LIN {X 0,Y 474.887,Z 291.332,A -85,B 0,C 180,E1 -7377.456,E2 -7377.456} C_VEL
LIN {X 0,Y 474.904,Z 291.328,A -85,B 0,C 180,E1 -7380,E2 -7380} C_VEL
LIN {X 0,Y 474.888,Z 291.326,A -85,B 0,C 180,E1 -7382.545,E2 -7382.545} C_VEL
LIN {X 0,Y 474.753,Z 291.35,A -85,B 0,C 180,E1 -7385.948,E2 -7385.948} C_VEL
LIN {X 0,Y 474.722,Z 291.348,A -85,B 0,C 180,E1 -7388.514,E2 -7388.514} C_VEL
LIN {X 0,Y 474.699,Z 291.357,A -85,B 0,C 180,E1 -7391.963,E2 -7391.963} C_VEL
LIN {X 0,Y 474.694,Z 291.35,A -85,B 0,C 180,E1 -7395.456,E2 -7395.456} C_VEL
LIN {X 0,Y 474.657,Z 291.355,A -85,B 0,C 180,E1 -7399.011,E2 -7399.011} C_VEL
LIN {X 0,Y 474.583,Z 291.365,A -85,B 0,C 180,E1 -7401.73,E2 -7401.73} C_VEL
LIN {X 0,Y 474.632,Z 291.365,A -85,B 0,C 180,E1 -7404.495,E2 -7404.495} C_VEL
LIN {X 0,Y 474.632,Z 291.357,A -85,B 0,C 180,E1 -7407.325,E2 -7407.325} C_VEL
LIN {X 0,Y 474.599,Z 291.366,A -85,B 0,C 180,E1 -7410.231,E2 -7410.231} C_VEL
LIN {X 0,Y 474.639,Z 291.358,A -85,B 0,C 180,E1 -7413.221,E2 -7413.221} C_VEL
LIN {X 0,Y 474.585,Z 291.367,A -85,B 0,C 180,E1 -7416.324,E2 -7416.324} C_VEL
LIN {X 0,Y 474.619,Z 291.359,A -85,B 0,C 180,E1 -7419.549,E2 -7419.549} C_VEL
LIN {X 0,Y 474.597,Z 291.363,A -85,B 0,C 180,E1 -7422.234,E2 -7422.234} C_VEL
LIN {X 0,Y 474.614,Z 291.364,A -85,B 0,C 180,E1 -7425.299,E2 -7425.299} C_VEL
LIN {X 0,Y 474.602,Z 291.361,A -85,B 0,C 180,E1 -7428.214,E2 -7428.214} C_VEL
LIN {X 0,Y 474.608,Z 291.363,A -85,B 0,C 180,E1 -7431.543,E2 -7431.543} C_VEL
LIN {X 0,Y 474.621,Z 291.361,A -85,B 0,C 180,E1 -7434.726,E2 -7434.726} C_VEL
LIN {X 0,Y 474.633,Z 291.359,A -85,B 0,C 180,E1 -7437.788,E2 -7437.788} C_VEL
LIN {X 0,Y 474.599,Z 291.364,A -85,B 0,C 180,E1 -7440.891,E2 -7440.891} C_VEL
LIN {X 0,Y 474.582,Z 291.37,A -85,B 0,C 180,E1 -7443.624,E2 -7443.624} C_VEL
LIN {X 0,Y 474.636,Z 291.357,A -85,B 0,C 180,E1 -7446.643,E2 -7446.643} C_VEL
LIN {X 0,Y 474.649,Z 291.358,A -85,B 0,C 180,E1 -7450.09,E2 -7450.09} C_VEL
LIN {X 0,Y 474.643,Z 291.361,A -85,B 0,C 180,E1 -7451.656,E2 -7451.656} C_VEL
LIN {X 0,Y 473.971,Z 291.446,A -85,B 0,C 180,E1 -7452.364,E2 -7452.364} C_VEL
LIN {X 0,Y 471.127,Z 291.8,A -85,B 0,C 180,E1 -7453.516,E2 -7453.516} C_VEL
LIN {X 0,Y 468.722,Z 292.097,A -85,B 0,C 180,E1 -7454.444,E2 -7454.444} C_VEL
LIN {X 0,Y 467.684,Z 292.224,A -85,B 0,C 180,E1 -7455.161,E2 -7455.161} C_VEL
LIN {X 0,Y 467.597,Z 292.235,A -85,B 0,C 180,E1 -7455.404,E2 -7455.404} C_VEL
LIN {X 0,Y 467.651,Z 292.236,A -85,B 0,C 180,E1 -7457.855,E2 -7457.855} C_VEL
LIN {X 0,Y 467.633,Z 292.231,A -85,B 0,C 180,E1 -7461.357,E2 -7461.357} C_VEL
LIN {X 0,Y 467.704,Z 292.229,A -85,B 0,C 180,E1 -7463.963,E2 -7463.963} C_VEL
LIN {X 0,Y 467.787,Z 292.211,A -85,B 0,C 180,E1 -7467.417,E2 -7467.417} C_VEL
LIN {X 0,Y 467.853,Z 292.208,A -85,B 0,C 180,E1 -7470.001,E2 -7470.001} C_VEL
LIN {X 0,Y 467.785,Z 292.214,A -85,B 0,C 180,E1 -7472.584,E2 -7472.584} C_VEL
LIN {X 0,Y 467.704,Z 292.225,A -85,B 0,C 180,E1 -7476.038,E2 -7476.038} C_VEL
LIN {X 0,Y 467.63,Z 292.235,A -85,B 0,C 180,E1 -7478.644,E2 -7478.644} C_VEL
LIN {X 0,Y 467.643,Z 292.234,A -85,B 0,C 180,E1 -7482.348,E2 -7482.348} C_VEL
LIN {X 0,Y 467.577,Z 292.237,A -85,B 0,C 180,E1 -7485.852,E2 -7485.852} C_VEL
LIN {X 0,Y 467.577,Z 292.245,A -85,B 0,C 180,E1 -7488.748,E2 -7488.748} C_VEL
LIN {X 0,Y 467.571,Z 292.242,A -85,B 0,C 180,E1 -7491.263,E2 -7491.263} C_VEL
LIN {X 0,Y 467.537,Z 292.245,A -85,B 0,C 180,E1 -7493.946,E2 -7493.946} C_VEL
LIN {X 0,Y 467.58,Z 292.359,A -85,B 0,C 180,E1 -7496.082,E2 -7496.082} C_VEL
LIN {X 0,Y 468.661,Z 298.553,A -85,B 0,C 180,E1 -7497.46,E2 -7497.46} C_VEL
LIN {X 0,Y 468.459,Z 309.115,A -85,B 0,C 180,E1 -7499.675,E2 -7499.675} C_VEL
LIN {X 0,Y 468.404,Z 311.167,A -85,B 0,C 180,E1 -7500.082,E2 -7500.082} C_VEL
LIN {X 0,Y 471.31,Z 326.35,A -85,B 0,C 180,E1 -7500.433,E2 -7500.433} C_VEL
LIN {X 0,Y 470.475,Z 418.507,A -85,B 0,C 180,E1 -7501.911,E2 -7501.911} C_VEL
LIN {X 0,Y 470.143,Z 431.815,A -85,B 0,C 180,E1 -7502.3,E2 -7502.3} C_VEL
LIN {X 0,Y 469.807,Z 444.646,A -85,B 0,C 180,E1 -7502.859,E2 -7502.859} C_VEL
LIN {X 0,Y 469.331,Z 456.478,A -85,B 0,C 180,E1 -7503.56,E2 -7503.56} C_VEL
LIN {X 0,Y 468.839,Z 468.329,A -85,B 0,C 180,E1 -7504.465,E2 -7504.465} C_VEL
LIN {X 0,Y 468.455,Z 478.228,A -85,B 0,C 180,E1 -7505.414,E2 -7505.414} C_VEL
LIN {X 0,Y 467.954,Z 487.6,A -85,B 0,C 180,E1 -7506.52,E2 -7506.52} C_VEL
LIN {X 0,Y 467.509,Z 496.556,A -85,B 0,C 180,E1 -7507.829,E2 -7507.829} C_VEL
LIN {X 0,Y 467.224,Z 503.935,A -85,B 0,C 180,E1 -7509.181,E2 -7509.181} C_VEL
LIN {X 0,Y 467.015,Z 508.97,A -85,B 0,C 180,E1 -7510.323,E2 -7510.323} C_VEL
LIN {X 0,Y 466.863,Z 513.083,A -85,B 0,C 180,E1 -7511.48,E2 -7511.48} C_VEL
LIN {X 0,Y 466.769,Z 516.363,A -85,B 0,C 180,E1 -7512.653,E2 -7512.653} C_VEL
LIN {X 0,Y 466.666,Z 518.873,A -85,B 0,C 180,E1 -7513.849,E2 -7513.849} C_VEL
LIN {X 0,Y 466.591,Z 520.607,A -85,B 0,C 180,E1 -7515.067,E2 -7515.067} C_VEL
LIN {X 0,Y 466.532,Z 521.536,A -85,B 0,C 180,E1 -7516.31,E2 -7516.31} C_VEL
LIN {X 0,Y 466.543,Z 521.611,A -85,B 0,C 180,E1 -7517.573,E2 -7517.573} C_VEL
LIN {X 0,Y 466.574,Z 520.813,A -85,B 0,C 180,E1 -7518.864,E2 -7518.864} C_VEL
LIN {X 0,Y 466.622,Z 519.065,A -85,B 0,C 180,E1 -7520.187,E2 -7520.187} C_VEL
LIN {X 0,Y 466.819,Z 515.392,A -85,B 0,C 180,E1 -7521.883,E2 -7521.883} C_VEL
LIN {X 0,Y 467.001,Z 510.099,A -85,B 0,C 180,E1 -7523.526,E2 -7523.526} C_VEL
LIN {X 0,Y 467.215,Z 504.977,A -85,B 0,C 180,E1 -7524.744,E2 -7524.744} C_VEL
LIN {X 0,Y 467.512,Z 498.452,A -85,B 0,C 180,E1 -7525.997,E2 -7525.997} C_VEL
LIN {X 0,Y 467.921,Z 490.267,A -85,B 0,C 180,E1 -7527.268,E2 -7527.268} C_VEL
LIN {X 0,Y 468.382,Z 480.754,A -85,B 0,C 180,E1 -7528.452,E2 -7528.452} C_VEL
LIN {X 0,Y 468.826,Z 470.415,A -85,B 0,C 180,E1 -7529.494,E2 -7529.494} C_VEL
LIN {X 0,Y 469.328,Z 459.314,A -85,B 0,C 180,E1 -7530.385,E2 -7530.385} C_VEL
LIN {X 0,Y 469.751,Z 447.055,A -85,B 0,C 180,E1 -7531.151,E2 -7531.151} C_VEL
LIN {X 0,Y 470.146,Z 434.659,A -85,B 0,C 180,E1 -7531.731,E2 -7531.731} C_VEL
LIN {X 0,Y 470.41,Z 422.487,A -85,B 0,C 180,E1 -7532.126,E2 -7532.126} C_VEL
LIN {X 0,Y 470.633,Z 405.056,A -85,B 0,C 180,E1 -7532.454,E2 -7532.454} C_VEL
LIN {X 0,Y 471.418,Z 326.13,A -85,B 0,C 180,E1 -7533.712,E2 -7533.712} C_VEL
LIN {X 0,Y 468.44,Z 310.387,A -85,B 0,C 180,E1 -7534.11,E2 -7534.11} C_VEL
LIN {X 0,Y 468.588,Z 297.583,A -85,B 0,C 180,E1 -7536.338,E2 -7536.338} C_VEL
LIN {X 0,Y 467.613,Z 292.241,A -85,B 0,C 180,E1 -7537.348,E2 -7537.348} C_VEL
LIN {X 0,Y 467.624,Z 292.236,A -85,B 0,C 180,E1 -7540.692,E2 -7540.692} C_VEL
LIN {X 0,Y 467.652,Z 292.233,A -85,B 0,C 180,E1 -7544.115,E2 -7544.115} C_VEL
LIN {X 0,Y 467.656,Z 292.235,A -85,B 0,C 180,E1 -7547.642,E2 -7547.642} C_VEL
LIN {X 0,Y 467.662,Z 292.228,A -85,B 0,C 180,E1 -7550.485,E2 -7550.485} C_VEL
LIN {X 0,Y 467.702,Z 292.224,A -85,B 0,C 180,E1 -7553.095,E2 -7553.095} C_VEL
LIN {X 0,Y 467.722,Z 292.221,A -85,B 0,C 180,E1 -7554.827,E2 -7554.827} C_VEL
LIN {X 0,Y 467.86,Z 292.206,A -85,B 0,C 180,E1 -7557.417,E2 -7557.417} C_VEL
LIN {X 0,Y 467.884,Z 292.205,A -85,B 0,C 180,E1 -7560,E2 -7560} C_VEL
LIN {X 0,Y 467.861,Z 292.204,A -85,B 0,C 180,E1 -7562.583,E2 -7562.583} C_VEL
LIN {X 0,Y 467.722,Z 292.226,A -85,B 0,C 180,E1 -7566.037,E2 -7566.037} C_VEL
LIN {X 0,Y 467.682,Z 292.227,A -85,B 0,C 180,E1 -7568.643,E2 -7568.643} C_VEL
LIN {X 0,Y 467.657,Z 292.233,A -85,B 0,C 180,E1 -7572.145,E2 -7572.145} C_VEL
LIN {X 0,Y 467.641,Z 292.23,A -85,B 0,C 180,E1 -7575.695,E2 -7575.695} C_VEL
LIN {X 0,Y 467.614,Z 292.238,A -85,B 0,C 180,E1 -7578.763,E2 -7578.763} C_VEL
LIN {X 0,Y 467.582,Z 292.236,A -85,B 0,C 180,E1 -7581.268,E2 -7581.268} C_VEL
LIN {X 0,Y 467.573,Z 292.237,A -85,B 0,C 180,E1 -7583.943,E2 -7583.943} C_VEL
LIN {X 0,Y 467.619,Z 292.238,A -85,B 0,C 180,E1 -7586.8,E2 -7586.8} C_VEL
LIN {X 0,Y 467.556,Z 292.24,A -85,B 0,C 180,E1 -7589.738,E2 -7589.738} C_VEL
LIN {X 0,Y 467.58,Z 292.24,A -85,B 0,C 180,E1 -7592.759,E2 -7592.759} C_VEL
LIN {X 0,Y 467.554,Z 292.241,A -85,B 0,C 180,E1 -7595.89,E2 -7595.89} C_VEL
LIN {X 0,Y 467.577,Z 292.244,A -85,B 0,C 180,E1 -7599.145,E2 -7599.145} C_VEL
LIN {X 0,Y 467.588,Z 292.238,A -85,B 0,C 180,E1 -7602.567,E2 -7602.567} C_VEL
LIN {X 0,Y 467.568,Z 292.244,A -85,B 0,C 180,E1 -7605.052,E2 -7605.052} C_VEL
LIN {X 0,Y 467.591,Z 292.243,A -85,B 0,C 180,E1 -7607.44,E2 -7607.44} C_VEL
LIN {X 0,Y 467.562,Z 292.241,A -85,B 0,C 180,E1 -7610.853,E2 -7610.853} C_VEL
LIN {X 0,Y 467.562,Z 292.245,A -85,B 0,C 180,E1 -7614.261,E2 -7614.261} C_VEL
LIN {X 0,Y 467.584,Z 292.244,A -85,B 0,C 180,E1 -7617.321,E2 -7617.321} C_VEL
LIN {X 0,Y 467.572,Z 292.241,A -85,B 0,C 180,E1 -7620.667,E2 -7620.667} C_VEL
LIN {X 0,Y 467.62,Z 292.239,A -85,B 0,C 180,E1 -7623.2,E2 -7623.2} C_VEL
LIN {X 0,Y 467.666,Z 292.395,A -85,B 0,C 180,E1 -7624.28,E2 -7624.28} C_VEL
LIN {X 0,Y 469.569,Z 302.744,A -85,B 0,C 180,E1 -7626.164,E2 -7626.164} C_VEL
LIN {X 0,Y 469.161,Z 316.935,A -85,B 0,C 180,E1 -7628.572,E2 -7628.572} C_VEL
LIN {X 0,Y 468.509,Z 336.543,A -85,B 0,C 180,E1 -7631.864,E2 -7631.864} C_VEL
LIN {X 0,Y 468.238,Z 342.994,A -85,B 0,C 180,E1 -7632.938,E2 -7632.938} C_VEL
LIN {X 0,Y 471.17,Z 362.703,A -85,B 0,C 180,E1 -7633.383,E2 -7633.383} C_VEL
LIN {X 0,Y 470.398,Z 451.756,A -85,B 0,C 180,E1 -7634.815,E2 -7634.815} C_VEL
LIN {X 0,Y 470.029,Z 464.941,A -85,B 0,C 180,E1 -7635.191,E2 -7635.191} C_VEL
LIN {X 0,Y 469.56,Z 478.23,A -85,B 0,C 180,E1 -7635.757,E2 -7635.757} C_VEL
LIN {X 0,Y 469.065,Z 490.218,A -85,B 0,C 180,E1 -7636.46,E2 -7636.46} C_VEL
LIN {X 0,Y 468.579,Z 502.383,A -85,B 0,C 180,E1 -7637.384,E2 -7637.384} C_VEL
LIN {X 0,Y 468.155,Z 512.119,A -85,B 0,C 180,E1 -7638.307,E2 -7638.307} C_VEL
LIN {X 0,Y 467.67,Z 521.451,A -85,B 0,C 180,E1 -7639.392,E2 -7639.392} C_VEL
LIN {X 0,Y 467.255,Z 530.522,A -85,B 0,C 180,E1 -7640.694,E2 -7640.694} C_VEL
LIN {X 0,Y 467.009,Z 537.837,A -85,B 0,C 180,E1 -7641.998,E2 -7641.998} C_VEL
LIN {X 0,Y 466.842,Z 542.78,A -85,B 0,C 180,E1 -7643.082,E2 -7643.082} C_VEL
LIN {X 0,Y 466.76,Z 547.587,A -85,B 0,C 180,E1 -7644.383,E2 -7644.383} C_VEL
LIN {X 0,Y 466.647,Z 551.26,A -85,B 0,C 180,E1 -7645.681,E2 -7645.681} C_VEL
LIN {X 0,Y 466.69,Z 553.16,A -85,B 0,C 180,E1 -7646.546,E2 -7646.546} C_VEL
LIN {X 0,Y 466.662,Z 554.584,A -85,B 0,C 180,E1 -7647.41,E2 -7647.41} C_VEL
LIN {X 0,Y 466.619,Z 556.227,A -85,B 0,C 180,E1 -7649.137,E2 -7649.137} C_VEL
LIN {X 0,Y 466.6,Z 556.451,A -85,B 0,C 180,E1 -7649.999,E2 -7649.999} C_VEL
LIN {X 0,Y 466.619,Z 556.237,A -85,B 0,C 180,E1 -7650.862,E2 -7650.862} C_VEL
LIN {X 0,Y 466.661,Z 554.626,A -85,B 0,C 180,E1 -7652.589,E2 -7652.589} C_VEL
LIN {X 0,Y 466.689,Z 553.211,A -85,B 0,C 180,E1 -7653.453,E2 -7653.453} C_VEL
LIN {X 0,Y 466.689,Z 550.24,A -85,B 0,C 180,E1 -7654.75,E2 -7654.75} C_VEL
LIN {X 0,Y 466.749,Z 546.214,A -85,B 0,C 180,E1 -7656.05,E2 -7656.05} C_VEL
LIN {X 0,Y 466.94,Z 540.011,A -85,B 0,C 180,E1 -7657.567,E2 -7657.567} C_VEL
LIN {X 0,Y 467.163,Z 533.24,A -85,B 0,C 180,E1 -7658.87,E2 -7658.87} C_VEL
LIN {X 0,Y 467.498,Z 524.835,A -85,B 0,C 180,E1 -7660.174,E2 -7660.174} C_VEL
LIN {X 0,Y 467.938,Z 516.177,A -85,B 0,C 180,E1 -7661.259,E2 -7661.259} C_VEL
LIN {X 0,Y 468.442,Z 505.997,A -85,B 0,C 180,E1 -7662.299,E2 -7662.299} C_VEL
LIN {X 0,Y 468.887,Z 494.923,A -85,B 0,C 180,E1 -7663.213,E2 -7663.213} C_VEL
LIN {X 0,Y 469.35,Z 483.182,A -85,B 0,C 180,E1 -7663.972,E2 -7663.972} C_VEL
LIN {X 0,Y 469.832,Z 470.995,A -85,B 0,C 180,E1 -7664.565,E2 -7664.565} C_VEL
LIN {X 0,Y 470.213,Z 457.736,A -85,B 0,C 180,E1 -7665.024,E2 -7665.024} C_VEL
LIN {X 0,Y 470.478,Z 443.027,A -85,B 0,C 180,E1 -7665.32,E2 -7665.32} C_VEL
LIN {X 0,Y 471.075,Z 362.031,A -85,B 0,C 180,E1 -7666.602,E2 -7666.602} C_VEL
LIN {X 0,Y 468.31,Z 343.777,A -85,B 0,C 180,E1 -7667.016,E2 -7667.016} C_VEL
LIN {X 0,Y 468.981,Z 326.897,A -85,B 0,C 180,E1 -7669.933,E2 -7669.933} C_VEL
LIN {X 0,Y 469.808,Z 309.995,A -85,B 0,C 180,E1 -7672.888,E2 -7672.888} C_VEL
LIN {X 0,Y 469.753,Z 303.092,A -85,B 0,C 180,E1 -7674.129,E2 -7674.129} C_VEL
LIN {X 0,Y 467.649,Z 292.236,A -85,B 0,C 180,E1 -7676.226,E2 -7676.226} C_VEL
LIN {X 0,Y 467.569,Z 292.24,A -85,B 0,C 180,E1 -7679.332,E2 -7679.332} C_VEL
LIN {X 0,Y 467.58,Z 292.239,A -85,B 0,C 180,E1 -7682.678,E2 -7682.678} C_VEL
LIN {X 0,Y 467.557,Z 292.241,A -85,B 0,C 180,E1 -7685.738,E2 -7685.738} C_VEL
LIN {X 0,Y 467.557,Z 292.239,A -85,B 0,C 180,E1 -7689.146,E2 -7689.146} C_VEL
LIN {X 0,Y 467.583,Z 292.242,A -85,B 0,C 180,E1 -7692.566,E2 -7692.566} C_VEL
LIN {X 0,Y 467.567,Z 292.239,A -85,B 0,C 180,E1 -7695.053,E2 -7695.053} C_VEL
LIN {X 0,Y 467.585,Z 292.235,A -85,B 0,C 180,E1 -7697.439,E2 -7697.439} C_VEL
LIN {X 0,Y 467.578,Z 292.242,A -85,B 0,C 180,E1 -7700.855,E2 -7700.855} C_VEL
LIN {X 0,Y 467.558,Z 292.241,A -85,B 0,C 180,E1 -7704.26,E2 -7704.26} C_VEL
LIN {X 0,Y 467.577,Z 292.239,A -85,B 0,C 180,E1 -7707.32,E2 -7707.32} C_VEL
LIN {X 0,Y 467.565,Z 292.243,A -85,B 0,C 180,E1 -7710.667,E2 -7710.667} C_VEL
LIN {X 0,Y 467.611,Z 292.238,A -85,B 0,C 180,E1 -7713.199,E2 -7713.199} C_VEL
LIN {X 0,Y 467.587,Z 292.236,A -85,B 0,C 180,E1 -7716.468,E2 -7716.468} C_VEL
LIN {X 0,Y 467.617,Z 292.233,A -85,B 0,C 180,E1 -7719.777,E2 -7719.777} C_VEL
LIN {X 0,Y 467.603,Z 292.234,A -85,B 0,C 180,E1 -7722.507,E2 -7722.507} C_VEL
LIN {X 0,Y 467.604,Z 292.24,A -85,B 0,C 180,E1 -7725.196,E2 -7725.196} C_VEL
LIN {X 0,Y 467.65,Z 292.23,A -85,B 0,C 180,E1 -7727.855,E2 -7727.855} C_VEL
LIN {X 0,Y 467.676,Z 292.231,A -85,B 0,C 180,E1 -7731.357,E2 -7731.357} C_VEL
LIN {X 0,Y 467.737,Z 292.219,A -85,B 0,C 180,E1 -7733.963,E2 -7733.963} C_VEL
LIN {X 0,Y 467.853,Z 292.207,A -85,B 0,C 180,E1 -7737.417,E2 -7737.417} C_VEL
LIN {X 0,Y 467.875,Z 292.204,A -85,B 0,C 180,E1 -7740,E2 -7740} C_VEL
LIN {X 0,Y 467.853,Z 292.202,A -85,B 0,C 180,E1 -7742.583,E2 -7742.583} C_VEL
LIN {X 0,Y 467.716,Z 292.226,A -85,B 0,C 180,E1 -7746.038,E2 -7746.038} C_VEL
LIN {X 0,Y 467.676,Z 292.225,A -85,B 0,C 180,E1 -7748.643,E2 -7748.643} C_VEL
LIN {X 0,Y 467.65,Z 292.235,A -85,B 0,C 180,E1 -7752.146,E2 -7752.146} C_VEL
LIN {X 0,Y 467.633,Z 292.232,A -85,B 0,C 180,E1 -7755.696,E2 -7755.696} C_VEL
LIN {X 0,Y 467.617,Z 292.231,A -85,B 0,C 180,E1 -7759.308,E2 -7759.308} C_VEL
LIN {X 0,Y 467.529,Z 292.247,A -85,B 0,C 180,E1 -7762.074,E2 -7762.074} C_VEL
LIN {X 0,Y 467.578,Z 292.238,A -85,B 0,C 180,E1 -7764.889,E2 -7764.889} C_VEL
LIN {X 0,Y 467.575,Z 292.237,A -85,B 0,C 180,E1 -7767.772,E2 -7767.772} C_VEL
LIN {X 0,Y 467.564,Z 292.24,A -85,B 0,C 180,E1 -7771.046,E2 -7771.046} C_VEL
LIN {X 0,Y 467.585,Z 292.238,A -85,B 0,C 180,E1 -7774.243,E2 -7774.243} C_VEL
LIN {X 0,Y 467.544,Z 292.243,A -85,B 0,C 180,E1 -7777.187,E2 -7777.187} C_VEL
LIN {X 0,Y 467.566,Z 292.239,A -85,B 0,C 180,E1 -7780.266,E2 -7780.266} C_VEL
LIN {X 0,Y 467.558,Z 292.243,A -85,B 0,C 180,E1 -7782.564,E2 -7782.564} C_VEL
LIN {X 0,Y 467.564,Z 292.245,A -85,B 0,C 180,E1 -7785.053,E2 -7785.053} C_VEL
LIN {X 0,Y 467.564,Z 292.242,A -85,B 0,C 180,E1 -7788.726,E2 -7788.726} C_VEL
LIN {X 0,Y 467.562,Z 292.238,A -85,B 0,C 180,E1 -7791.956,E2 -7791.956} C_VEL
LIN {X 0,Y 467.558,Z 292.247,A -85,B 0,C 180,E1 -7795.168,E2 -7795.168} C_VEL
LIN {X 0,Y 467.58,Z 292.236,A -85,B 0,C 180,E1 -7798.261,E2 -7798.261} C_VEL
LIN {X 0,Y 467.546,Z 292.247,A -85,B 0,C 180,E1 -7801.249,E2 -7801.249} C_VEL
LIN {X 0,Y 467.577,Z 292.236,A -85,B 0,C 180,E1 -7804.402,E2 -7804.402} C_VEL
LIN {X 0,Y 467.578,Z 292.238,A -85,B 0,C 180,E1 -7806.997,E2 -7806.997} C_VEL
LIN {X 0,Y 467.62,Z 292.237,A -85,B 0,C 180,E1 -7809.778,E2 -7809.778} C_VEL
LIN {X 0,Y 467.589,Z 292.235,A -85,B 0,C 180,E1 -7812.507,E2 -7812.507} C_VEL
LIN {X 0,Y 467.597,Z 292.235,A -85,B 0,C 180,E1 -7815.404,E2 -7815.404} C_VEL
LIN {X 0,Y 466.924,Z 292.322,A -85,B 0,C 180,E1 -7816.123,E2 -7816.123} C_VEL
LIN {X 0,Y 464.076,Z 292.674,A -85,B 0,C 180,E1 -7817.291,E2 -7817.291} C_VEL
LIN {X 0,Y 461.671,Z 292.975,A -85,B 0,C 180,E1 -7818.233,E2 -7818.233} C_VEL
LIN {X 0,Y 460.638,Z 293.101,A -85,B 0,C 180,E1 -7818.961,E2 -7818.961} C_VEL
LIN {X 0,Y 460.553,Z 293.112,A -85,B 0,C 180,E1 -7819.207,E2 -7819.207} C_VEL
LIN {X 0,Y 460.667,Z 293.098,A -85,B 0,C 180,E1 -7822.595,E2 -7822.595} C_VEL
LIN {X 0,Y 460.676,Z 293.097,A -85,B 0,C 180,E1 -7824.749,E2 -7824.749} C_VEL
LIN {X 0,Y 460.718,Z 293.098,A -85,B 0,C 180,E1 -7828.252,E2 -7828.252} C_VEL
LIN {X 0,Y 460.822,Z 293.084,A -85,B 0,C 180,E1 -7830.001,E2 -7830.001} C_VEL
LIN {X 0,Y 460.732,Z 293.092,A -85,B 0,C 180,E1 -7832.623,E2 -7832.623} C_VEL
LIN {X 0,Y 460.67,Z 293.102,A -85,B 0,C 180,E1 -7836.131,E2 -7836.131} C_VEL
LIN {X 0,Y 460.584,Z 293.111,A -85,B 0,C 180,E1 -7838.777,E2 -7838.777} C_VEL
LIN {X 0,Y 460.602,Z 293.113,A -85,B 0,C 180,E1 -7842.435,E2 -7842.435} C_VEL
LIN {X 0,Y 460.531,Z 293.115,A -85,B 0,C 180,E1 -7845.965,E2 -7845.965} C_VEL
LIN {X 0,Y 460.535,Z 293.121,A -85,B 0,C 180,E1 -7848.887,E2 -7848.887} C_VEL
LIN {X 0,Y 460.516,Z 293.119,A -85,B 0,C 180,E1 -7851.486,E2 -7851.486} C_VEL
LIN {X 0,Y 460.5,Z 293.124,A -85,B 0,C 180,E1 -7854.335,E2 -7854.335} C_VEL
LIN {X 0,Y 460.551,Z 293.198,A -85,B 0,C 180,E1 -7855.904,E2 -7855.904} C_VEL
LIN {X 0,Y 461.786,Z 300.731,A -85,B 0,C 180,E1 -7857.593,E2 -7857.593} C_VEL
LIN {X 0,Y 461.463,Z 311.503,A -85,B 0,C 180,E1 -7859.83,E2 -7859.83} C_VEL
LIN {X 0,Y 464.48,Z 327.191,A -85,B 0,C 180,E1 -7860.203,E2 -7860.203} C_VEL
LIN {X 0,Y 463.601,Z 418.569,A -85,B 0,C 180,E1 -7861.692,E2 -7861.692} C_VEL
LIN {X 0,Y 463.247,Z 431.996,A -85,B 0,C 180,E1 -7862.089,E2 -7862.089} C_VEL
LIN {X 0,Y 462.943,Z 443.935,A -85,B 0,C 180,E1 -7862.611,E2 -7862.611} C_VEL
LIN {X 0,Y 462.456,Z 455.653,A -85,B 0,C 180,E1 -7863.296,E2 -7863.296} C_VEL
LIN {X 0,Y 461.964,Z 466.743,A -85,B 0,C 180,E1 -7864.132,E2 -7864.132} C_VEL
LIN {X 0,Y 461.501,Z 477.687,A -85,B 0,C 180,E1 -7865.168,E2 -7865.168} C_VEL
LIN {X 0,Y 461.043,Z 486.998,A -85,B 0,C 180,E1 -7866.26,E2 -7866.26} C_VEL
LIN {X 0,Y 460.569,Z 495.479,A -85,B 0,C 180,E1 -7867.487,E2 -7867.487} C_VEL
LIN {X 0,Y 460.21,Z 503.066,A -85,B 0,C 180,E1 -7868.845,E2 -7868.845} C_VEL
LIN {X 0,Y 459.948,Z 509.024,A -85,B 0,C 180,E1 -7870.181,E2 -7870.181} C_VEL
LIN {X 0,Y 459.786,Z 513.638,A -85,B 0,C 180,E1 -7871.497,E2 -7871.497} C_VEL
LIN {X 0,Y 459.67,Z 517.091,A -85,B 0,C 180,E1 -7872.786,E2 -7872.786} C_VEL
LIN {X 0,Y 459.552,Z 519.529,A -85,B 0,C 180,E1 -7874.046,E2 -7874.046} C_VEL
LIN {X 0,Y 459.484,Z 521.091,A -85,B 0,C 180,E1 -7875.284,E2 -7875.284} C_VEL
LIN {X 0,Y 459.438,Z 521.856,A -85,B 0,C 180,E1 -7876.499,E2 -7876.499} C_VEL
LIN {X 0,Y 459.447,Z 521.859,A -85,B 0,C 180,E1 -7877.696,E2 -7877.696} C_VEL
LIN {X 0,Y 459.485,Z 521.102,A -85,B 0,C 180,E1 -7878.875,E2 -7878.875} C_VEL
LIN {X 0,Y 459.53,Z 519.676,A -85,B 0,C 180,E1 -7880.033,E2 -7880.033} C_VEL
LIN {X 0,Y 459.649,Z 517.422,A -85,B 0,C 180,E1 -7881.241,E2 -7881.241} C_VEL
LIN {X 0,Y 459.819,Z 513.752,A -85,B 0,C 180,E1 -7882.635,E2 -7882.635} C_VEL
LIN {X 0,Y 460.028,Z 508.693,A -85,B 0,C 180,E1 -7884.067,E2 -7884.067} C_VEL
LIN {X 0,Y 460.36,Z 501.626,A -85,B 0,C 180,E1 -7885.607,E2 -7885.607} C_VEL
LIN {X 0,Y 460.813,Z 493.323,A -85,B 0,C 180,E1 -7887.016,E2 -7887.016} C_VEL
LIN {X 0,Y 461.253,Z 484.363,A -85,B 0,C 180,E1 -7888.235,E2 -7888.235} C_VEL
LIN {X 0,Y 461.72,Z 474.342,A -85,B 0,C 180,E1 -7889.341,E2 -7889.341} C_VEL
LIN {X 0,Y 462.234,Z 463.584,A -85,B 0,C 180,E1 -7890.287,E2 -7890.287} C_VEL
LIN {X 0,Y 462.769,Z 451.178,A -85,B 0,C 180,E1 -7891.146,E2 -7891.146} C_VEL
LIN {X 0,Y 463.192,Z 439.482,A -85,B 0,C 180,E1 -7891.76,E2 -7891.76} C_VEL
LIN {X 0,Y 463.466,Z 425.92,A -85,B 0,C 180,E1 -7892.267,E2 -7892.267} C_VEL
LIN {X 0,Y 463.76,Z 412.27,A -85,B 0,C 180,E1 -7892.577,E2 -7892.577} C_VEL
LIN {X 0,Y 464.586,Z 326.297,A -85,B 0,C 180,E1 -7893.979,E2 -7893.979} C_VEL
LIN {X 0,Y 461.528,Z 310.691,A -85,B 0,C 180,E1 -7894.378,E2 -7894.378} C_VEL
LIN {X 0,Y 461.687,Z 299.498,A -85,B 0,C 180,E1 -7896.34,E2 -7896.34} C_VEL
LIN {X 0,Y 460.556,Z 293.119,A -85,B 0,C 180,E1 -7897.544,E2 -7897.544} C_VEL
LIN {X 0,Y 460.571,Z 293.113,A -85,B 0,C 180,E1 -7900.384,E2 -7900.384} C_VEL
LIN {X 0,Y 460.603,Z 293.112,A -85,B 0,C 180,E1 -7904.002,E2 -7904.002} C_VEL
LIN {X 0,Y 460.611,Z 293.112,A -85,B 0,C 180,E1 -7907.666,E2 -7907.666} C_VEL
LIN {X 0,Y 460.628,Z 293.107,A -85,B 0,C 180,E1 -7911.224,E2 -7911.224} C_VEL
LIN {X 0,Y 460.702,Z 293.1,A -85,B 0,C 180,E1 -7913.87,E2 -7913.87} C_VEL
LIN {X 0,Y 460.801,Z 293.085,A -85,B 0,C 180,E1 -7917.377,E2 -7917.377} C_VEL
LIN {X 0,Y 460.854,Z 293.081,A -85,B 0,C 180,E1 -7920,E2 -7920} C_VEL
LIN {X 0,Y 460.802,Z 293.083,A -85,B 0,C 180,E1 -7922.622,E2 -7922.622} C_VEL
LIN {X 0,Y 460.686,Z 293.101,A -85,B 0,C 180,E1 -7926.13,E2 -7926.13} C_VEL
LIN {X 0,Y 460.629,Z 293.104,A -85,B 0,C 180,E1 -7928.776,E2 -7928.776} C_VEL
LIN {X 0,Y 460.615,Z 293.109,A -85,B 0,C 180,E1 -7932.445,E2 -7932.445} C_VEL
LIN {X 0,Y 460.602,Z 293.109,A -85,B 0,C 180,E1 -7935.997,E2 -7935.997} C_VEL
LIN {X 0,Y 460.569,Z 293.11,A -85,B 0,C 180,E1 -7939.615,E2 -7939.615} C_VEL
LIN {X 0,Y 460.512,Z 293.121,A -85,B 0,C 180,E1 -7942.429,E2 -7942.429} C_VEL
LIN {X 0,Y 460.569,Z 293.109,A -85,B 0,C 180,E1 -7945.802,E2 -7945.802} C_VEL
LIN {X 0,Y 460.554,Z 293.109,A -85,B 0,C 180,E1 -7948.233,E2 -7948.233} C_VEL
LIN {X 0,Y 460.522,Z 293.118,A -85,B 0,C 180,E1 -7951.283,E2 -7951.283} C_VEL
LIN {X 0,Y 460.524,Z 293.117,A -85,B 0,C 180,E1 -7954.504,E2 -7954.504} C_VEL
LIN {X 0,Y 460.503,Z 293.119,A -85,B 0,C 180,E1 -7957.623,E2 -7957.623} C_VEL
LIN {X 0,Y 460.541,Z 293.113,A -85,B 0,C 180,E1 -7960.269,E2 -7960.269} C_VEL
LIN {X 0,Y 460.501,Z 293.124,A -85,B 0,C 180,E1 -7963.375,E2 -7963.375} C_VEL
LIN {X 0,Y 460.5,Z 293.12,A -85,B 0,C 180,E1 -7966.624,E2 -7966.624} C_VEL
LIN {X 0,Y 460.541,Z 293.119,A -85,B 0,C 180,E1 -7969.731,E2 -7969.731} C_VEL
LIN {X 0,Y 460.502,Z 293.122,A -85,B 0,C 180,E1 -7972.524,E2 -7972.524} C_VEL
LIN {X 0,Y 460.549,Z 293.123,A -85,B 0,C 180,E1 -7975.624,E2 -7975.624} C_VEL
LIN {X 0,Y 460.54,Z 293.117,A -85,B 0,C 180,E1 -7978.744,E2 -7978.744} C_VEL
LIN {X 0,Y 460.584,Z 293.116,A -85,B 0,C 180,E1 -7982.254,E2 -7982.254} C_VEL
LIN {X 0,Y 460.614,Z 293.192,A -85,B 0,C 180,E1 -7984.045,E2 -7984.045} C_VEL
LIN {X 0,Y 462.538,Z 303.263,A -85,B 0,C 180,E1 -7985.922,E2 -7985.922} C_VEL
LIN {X 0,Y 462.622,Z 307.903,A -85,B 0,C 180,E1 -7986.735,E2 -7986.735} C_VEL
LIN {X 0,Y 461.894,Z 326.853,A -85,B 0,C 180,E1 -7989.979,E2 -7989.979} C_VEL
LIN {X 0,Y 461.277,Z 342.723,A -85,B 0,C 180,E1 -7992.666,E2 -7992.666} C_VEL
LIN {X 0,Y 464.368,Z 363.157,A -85,B 0,C 180,E1 -7993.133,E2 -7993.133} C_VEL
LIN {X 0,Y 463.564,Z 451.556,A -85,B 0,C 180,E1 -7994.586,E2 -7994.586} C_VEL
LIN {X 0,Y 463.176,Z 464.703,A -85,B 0,C 180,E1 -7994.967,E2 -7994.967} C_VEL
LIN {X 0,Y 462.658,Z 477.976,A -85,B 0,C 180,E1 -7995.54,E2 -7995.54} C_VEL
LIN {X 0,Y 462.145,Z 489.957,A -85,B 0,C 180,E1 -7996.254,E2 -7996.254} C_VEL
LIN {X 0,Y 461.66,Z 501.506,A -85,B 0,C 180,E1 -7997.139,E2 -7997.139} C_VEL
LIN {X 0,Y 461.183,Z 511.858,A -85,B 0,C 180,E1 -7998.127,E2 -7998.127} C_VEL
LIN {X 0,Y 460.639,Z 521.188,A -85,B 0,C 180,E1 -7999.228,E2 -7999.228} C_VEL
LIN {X 0,Y 460.209,Z 530.262,A -85,B 0,C 180,E1 -8000.551,E2 -8000.551} C_VEL
LIN {X 0,Y 459.95,Z 537.579,A -85,B 0,C 180,E1 -8001.874,E2 -8001.874} C_VEL
LIN {X 0,Y 459.74,Z 543.711,A -85,B 0,C 180,E1 -8003.272,E2 -8003.272} C_VEL
LIN {X 0,Y 459.65,Z 548.66,A -85,B 0,C 180,E1 -8004.736,E2 -8004.736} C_VEL
LIN {X 0,Y 459.565,Z 550.995,A -85,B 0,C 180,E1 -8005.614,E2 -8005.614} C_VEL
LIN {X 0,Y 459.585,Z 552.895,A -85,B 0,C 180,E1 -8006.493,E2 -8006.493} C_VEL
LIN {X 0,Y 459.584,Z 554.32,A -85,B 0,C 180,E1 -8007.37,E2 -8007.37} C_VEL
LIN {X 0,Y 459.552,Z 555.964,A -85,B 0,C 180,E1 -8009.123,E2 -8009.123} C_VEL
LIN {X 0,Y 459.532,Z 556.188,A -85,B 0,C 180,E1 -8009.999,E2 -8009.999} C_VEL
LIN {X 0,Y 459.552,Z 555.973,A -85,B 0,C 180,E1 -8010.876,E2 -8010.876} C_VEL
LIN {X 0,Y 459.584,Z 554.358,A -85,B 0,C 180,E1 -8012.629,E2 -8012.629} C_VEL
LIN {X 0,Y 459.585,Z 552.939,A -85,B 0,C 180,E1 -8013.506,E2 -8013.506} C_VEL
LIN {X 0,Y 459.616,Z 549.964,A -85,B 0,C 180,E1 -8014.824,E2 -8014.824} C_VEL
LIN {X 0,Y 459.713,Z 544.874,A -85,B 0,C 180,E1 -8016.43,E2 -8016.43} C_VEL
LIN {X 0,Y 459.889,Z 538.69,A -85,B 0,C 180,E1 -8017.905,E2 -8017.905} C_VEL
LIN {X 0,Y 460.175,Z 531.667,A -85,B 0,C 180,E1 -8019.227,E2 -8019.227} C_VEL
LIN {X 0,Y 460.557,Z 522.856,A -85,B 0,C 180,E1 -8020.551,E2 -8020.551} C_VEL
LIN {X 0,Y 461.119,Z 512.851,A -85,B 0,C 180,E1 -8021.762,E2 -8021.762} C_VEL
LIN {X 0,Y 461.561,Z 502.918,A -85,B 0,C 180,E1 -8022.732,E2 -8022.732} C_VEL
LIN {X 0,Y 462.069,Z 491.349,A -85,B 0,C 180,E1 -8023.635,E2 -8023.635} C_VEL
LIN {X 0,Y 462.561,Z 479.647,A -85,B 0,C 180,E1 -8024.349,E2 -8024.349} C_VEL
LIN {X 0,Y 463.046,Z 466.974,A -85,B 0,C 180,E1 -8024.924,E2 -8024.924} C_VEL
LIN {X 0,Y 463.466,Z 453.581,A -85,B 0,C 180,E1 -8025.332,E2 -8025.332} C_VEL
LIN {X 0,Y 463.809,Z 421.729,A -85,B 0,C 180,E1 -8025.871,E2 -8025.871} C_VEL
LIN {X 0,Y 464.197,Z 362.391,A -85,B 0,C 180,E1 -8026.833,E2 -8026.833} C_VEL
LIN {X 0,Y 461.324,Z 343.668,A -85,B 0,C 180,E1 -8027.249,E2 -8027.249} C_VEL
LIN {X 0,Y 462.074,Z 326.606,A -85,B 0,C 180,E1 -8030.243,E2 -8030.243} C_VEL
LIN {X 0,Y 462.965,Z 308.418,A -85,B 0,C 180,E1 -8033.483,E2 -8033.483} C_VEL
LIN {X 0,Y 462.61,Z 303.188,A -85,B 0,C 180,E1 -8034.454,E2 -8034.454} C_VEL
LIN {X 0,Y 460.587,Z 293.114,A -85,B 0,C 180,E1 -8036.446,E2 -8036.446} C_VEL
LIN {X 0,Y 460.53,Z 293.119,A -85,B 0,C 180,E1 -8039.558,E2 -8039.558} C_VEL
LIN {X 0,Y 460.53,Z 293.124,A -85,B 0,C 180,E1 -8042.284,E2 -8042.284} C_VEL
LIN {X 0,Y 460.508,Z 293.117,A -85,B 0,C 180,E1 -8045.445,E2 -8045.445} C_VEL
LIN {X 0,Y 460.531,Z 293.116,A -85,B 0,C 180,E1 -8048.895,E2 -8048.895} C_VEL
LIN {X 0,Y 460.519,Z 293.121,A -85,B 0,C 180,E1 -8052.181,E2 -8052.181} C_VEL
LIN {X 0,Y 460.517,Z 293.116,A -85,B 0,C 180,E1 -8055.411,E2 -8055.411} C_VEL
LIN {X 0,Y 460.531,Z 293.12,A -85,B 0,C 180,E1 -8058.396,E2 -8058.396} C_VEL
LIN {X 0,Y 460.523,Z 293.116,A -85,B 0,C 180,E1 -8061.267,E2 -8061.267} C_VEL
LIN {X 0,Y 460.508,Z 293.123,A -85,B 0,C 180,E1 -8064.554,E2 -8064.554} C_VEL
LIN {X 0,Y 460.527,Z 293.115,A -85,B 0,C 180,E1 -8067.715,E2 -8067.715} C_VEL
LIN {X 0,Y 460.535,Z 293.12,A -85,B 0,C 180,E1 -8070.769,E2 -8070.769} C_VEL
LIN {X 0,Y 460.558,Z 293.111,A -85,B 0,C 180,E1 -8073.734,E2 -8073.734} C_VEL
LIN {X 0,Y 460.54,Z 293.115,A -85,B 0,C 180,E1 -8076.624,E2 -8076.624} C_VEL
LIN {X 0,Y 460.545,Z 293.117,A -85,B 0,C 180,E1 -8079.453,E2 -8079.453} C_VEL
LIN {X 0,Y 460.553,Z 293.111,A -85,B 0,C 180,E1 -8082.23,E2 -8082.23} C_VEL
LIN {X 0,Y 460.562,Z 293.114,A -85,B 0,C 180,E1 -8084.965,E2 -8084.965} C_VEL
LIN {X 0,Y 460.605,Z 293.105,A -85,B 0,C 180,E1 -8088.559,E2 -8088.559} C_VEL
LIN {X 0,Y 460.689,Z 293.096,A -85,B 0,C 180,E1 -8092.109,E2 -8092.109} C_VEL
LIN {X 0,Y 460.69,Z 293.094,A -85,B 0,C 180,E1 -8094.748,E2 -8094.748} C_VEL
LIN {X 0,Y 460.793,Z 293.086,A -85,B 0,C 180,E1 -8097.378,E2 -8097.378} C_VEL
LIN {X 0,Y 460.845,Z 293.08,A -85,B 0,C 180,E1 -8100,E2 -8100} C_VEL
LIN {X 0,Y 460.794,Z 293.081,A -85,B 0,C 180,E1 -8102.623,E2 -8102.623} C_VEL
LIN {X 0,Y 460.68,Z 293.101,A -85,B 0,C 180,E1 -8106.131,E2 -8106.131} C_VEL
LIN {X 0,Y 460.623,Z 293.103,A -85,B 0,C 180,E1 -8108.777,E2 -8108.777} C_VEL
LIN {X 0,Y 460.608,Z 293.108,A -85,B 0,C 180,E1 -8112.445,E2 -8112.445} C_VEL
LIN {X 0,Y 460.595,Z 293.112,A -85,B 0,C 180,E1 -8115.998,E2 -8115.998} C_VEL
LIN {X 0,Y 460.563,Z 293.111,A -85,B 0,C 180,E1 -8119.616,E2 -8119.616} C_VEL
LIN {X 0,Y 460.506,Z 293.125,A -85,B 0,C 180,E1 -8122.429,E2 -8122.429} C_VEL
LIN {X 0,Y 460.544,Z 293.114,A -85,B 0,C 180,E1 -8125.798,E2 -8125.798} C_VEL
LIN {X 0,Y 460.522,Z 293.12,A -85,B 0,C 180,E1 -8128.235,E2 -8128.235} C_VEL
LIN {X 0,Y 460.517,Z 293.116,A -85,B 0,C 180,E1 -8131.284,E2 -8131.284} C_VEL
LIN {X 0,Y 460.528,Z 293.121,A -85,B 0,C 180,E1 -8134.506,E2 -8134.506} C_VEL
LIN {X 0,Y 460.497,Z 293.118,A -85,B 0,C 180,E1 -8137.624,E2 -8137.624} C_VEL
LIN {X 0,Y 460.531,Z 293.116,A -85,B 0,C 180,E1 -8140.269,E2 -8140.269} C_VEL
LIN {X 0,Y 460.506,Z 293.12,A -85,B 0,C 180,E1 -8143.375,E2 -8143.375} C_VEL
LIN {X 0,Y 460.501,Z 293.121,A -85,B 0,C 180,E1 -8146.626,E2 -8146.626} C_VEL
LIN {X 0,Y 460.523,Z 293.116,A -85,B 0,C 180,E1 -8149.734,E2 -8149.734} C_VEL
LIN {X 0,Y 460.498,Z 293.119,A -85,B 0,C 180,E1 -8152.525,E2 -8152.525} C_VEL
LIN {X 0,Y 460.537,Z 293.117,A -85,B 0,C 180,E1 -8155.624,E2 -8155.624} C_VEL
LIN {X 0,Y 460.521,Z 293.117,A -85,B 0,C 180,E1 -8158.744,E2 -8158.744} C_VEL
LIN {X 0,Y 460.508,Z 293.12,A -85,B 0,C 180,E1 -8161.765,E2 -8161.765} C_VEL
LIN {X 0,Y 460.521,Z 293.116,A -85,B 0,C 180,E1 -8164.704,E2 -8164.704} C_VEL
LIN {X 0,Y 460.513,Z 293.125,A -85,B 0,C 180,E1 -8167.572,E2 -8167.572} C_VEL
LIN {X 0,Y 460.567,Z 293.11,A -85,B 0,C 180,E1 -8170.385,E2 -8170.385} C_VEL
LIN {X 0,Y 460.582,Z 293.112,A -85,B 0,C 180,E1 -8174.013,E2 -8174.013} C_VEL
LIN {X 0,Y 460.606,Z 293.111,A -85,B 0,C 180,E1 -8177.666,E2 -8177.666} C_VEL
LIN {X 0,Y 460.553,Z 293.112,A -85,B 0,C 180,E1 -8179.207,E2 -8179.207} C_VEL
LIN {X 0,Y 459.887,Z 293.203,A -85,B 0,C 180,E1 -8179.937,E2 -8179.937} C_VEL
LIN {X 0,Y 457.056,Z 293.55,A -85,B 0,C 180,E1 -8181.123,E2 -8181.123} C_VEL
LIN {X 0,Y 454.674,Z 293.851,A -85,B 0,C 180,E1 -8182.08,E2 -8182.08} C_VEL
LIN {X 0,Y 453.664,Z 293.97,A -85,B 0,C 180,E1 -8182.819,E2 -8182.819} C_VEL
LIN {X 0,Y 453.589,Z 293.979,A -85,B 0,C 180,E1 -8183.069,E2 -8183.069} C_VEL
LIN {X 0,Y 453.649,Z 293.972,A -85,B 0,C 180,E1 -8184.667,E2 -8184.667} C_VEL
LIN {X 0,Y 453.688,Z 293.974,A -85,B 0,C 180,E1 -8188.225,E2 -8188.225} C_VEL
LIN {X 0,Y 453.771,Z 293.962,A -85,B 0,C 180,E1 -8190.001,E2 -8190.001} C_VEL
LIN {X 0,Y 453.681,Z 293.97,A -85,B 0,C 180,E1 -8192.664,E2 -8192.664} C_VEL
LIN {X 0,Y 453.638,Z 293.98,A -85,B 0,C 180,E1 -8196.226,E2 -8196.226} C_VEL
LIN {X 0,Y 453.554,Z 293.985,A -85,B 0,C 180,E1 -8198.915,E2 -8198.915} C_VEL
LIN {X 0,Y 453.57,Z 293.99,A -85,B 0,C 180,E1 -8202.529,E2 -8202.529} C_VEL
LIN {X 0,Y 453.495,Z 293.993,A -85,B 0,C 180,E1 -8206.198,E2 -8206.198} C_VEL
LIN {X 0,Y 453.49,Z 293.997,A -85,B 0,C 180,E1 -8209.028,E2 -8209.028} C_VEL
LIN {X 0,Y 453.475,Z 293.996,A -85,B 0,C 180,E1 -8211.837,E2 -8211.837} C_VEL
LIN {X 0,Y 453.475,Z 294.001,A -85,B 0,C 180,E1 -8215.227,E2 -8215.227} C_VEL
LIN {X 0,Y 453.493,Z 294.029,A -85,B 0,C 180,E1 -8215.718,E2 -8215.718} C_VEL
LIN {X 0,Y 454.762,Z 301.294,A -85,B 0,C 180,E1 -8217.372,E2 -8217.372} C_VEL
LIN {X 0,Y 454.5,Z 311.538,A -85,B 0,C 180,E1 -8219.563,E2 -8219.563} C_VEL
LIN {X 0,Y 457.678,Z 328.34,A -85,B 0,C 180,E1 -8219.973,E2 -8219.973} C_VEL
LIN {X 0,Y 456.74,Z 419.157,A -85,B 0,C 180,E1 -8221.481,E2 -8221.481} C_VEL
LIN {X 0,Y 456.359,Z 432.62,A -85,B 0,C 180,E1 -8221.888,E2 -8221.888} C_VEL
LIN {X 0,Y 456.048,Z 444.203,A -85,B 0,C 180,E1 -8222.406,E2 -8222.406} C_VEL
LIN {X 0,Y 455.517,Z 456.548,A -85,B 0,C 180,E1 -8223.145,E2 -8223.145} C_VEL
LIN {X 0,Y 454.955,Z 468.228,A -85,B 0,C 180,E1 -8224.055,E2 -8224.055} C_VEL
LIN {X 0,Y 454.544,Z 477.636,A -85,B 0,C 180,E1 -8224.968,E2 -8224.968} C_VEL
LIN {X 0,Y 454.048,Z 486.658,A -85,B 0,C 180,E1 -8226.029,E2 -8226.029} C_VEL
LIN {X 0,Y 453.619,Z 494.647,A -85,B 0,C 180,E1 -8227.174,E2 -8227.174} C_VEL
LIN {X 0,Y 453.235,Z 502.32,A -85,B 0,C 180,E1 -8228.532,E2 -8228.532} C_VEL
LIN {X 0,Y 452.895,Z 508.934,A -85,B 0,C 180,E1 -8230.002,E2 -8230.002} C_VEL
LIN {X 0,Y 452.732,Z 513.344,A -85,B 0,C 180,E1 -8231.251,E2 -8231.251} C_VEL
LIN {X 0,Y 452.625,Z 516.763,A -85,B 0,C 180,E1 -8232.488,E2 -8232.488} C_VEL
LIN {X 0,Y 452.486,Z 519.318,A -85,B 0,C 180,E1 -8233.723,E2 -8233.723} C_VEL
LIN {X 0,Y 452.439,Z 520.36,A -85,B 0,C 180,E1 -8234.393,E2 -8234.393} C_VEL
LIN {X 0,Y 452.387,Z 521.693,A -85,B 0,C 180,E1 -8235.645,E2 -8235.645} C_VEL
LIN {X 0,Y 452.342,Z 522.201,A -85,B 0,C 180,E1 -8236.906,E2 -8236.906} C_VEL
LIN {X 0,Y 452.37,Z 521.882,A -85,B 0,C 180,E1 -8238.222,E2 -8238.222} C_VEL
LIN {X 0,Y 452.395,Z 520.652,A -85,B 0,C 180,E1 -8239.572,E2 -8239.572} C_VEL
LIN {X 0,Y 452.529,Z 518.435,A -85,B 0,C 180,E1 -8240.944,E2 -8240.944} C_VEL
LIN {X 0,Y 452.719,Z 515.101,A -85,B 0,C 180,E1 -8242.347,E2 -8242.347} C_VEL
LIN {X 0,Y 452.925,Z 510.179,A -85,B 0,C 180,E1 -8243.868,E2 -8243.868} C_VEL
LIN {X 0,Y 453.216,Z 504.246,A -85,B 0,C 180,E1 -8245.273,E2 -8245.273} C_VEL
LIN {X 0,Y 453.523,Z 497.968,A -85,B 0,C 180,E1 -8246.468,E2 -8246.468} C_VEL
LIN {X 0,Y 453.983,Z 489.904,A -85,B 0,C 180,E1 -8247.718,E2 -8247.718} C_VEL
LIN {X 0,Y 454.508,Z 480.263,A -85,B 0,C 180,E1 -8248.93,E2 -8248.93} C_VEL
LIN {X 0,Y 454.984,Z 470.963,A -85,B 0,C 180,E1 -8249.885,E2 -8249.885} C_VEL
LIN {X 0,Y 455.554,Z 459.929,A -85,B 0,C 180,E1 -8250.798,E2 -8250.798} C_VEL
LIN {X 0,Y 456.024,Z 448.262,A -85,B 0,C 180,E1 -8251.554,E2 -8251.554} C_VEL
LIN {X 0,Y 456.465,Z 435.467,A -85,B 0,C 180,E1 -8252.179,E2 -8252.179} C_VEL
LIN {X 0,Y 456.781,Z 422.76,A -85,B 0,C 180,E1 -8252.604,E2 -8252.604} C_VEL
LIN {X 0,Y 457.021,Z 405.311,A -85,B 0,C 180,E1 -8252.942,E2 -8252.942} C_VEL
LIN {X 0,Y 457.819,Z 327.03,A -85,B 0,C 180,E1 -8254.242,E2 -8254.242} C_VEL
LIN {X 0,Y 454.617,Z 310.814,A -85,B 0,C 180,E1 -8254.688,E2 -8254.688} C_VEL
LIN {X 0,Y 454.729,Z 300.361,A -85,B 0,C 180,E1 -8256.548,E2 -8256.548} C_VEL
LIN {X 0,Y 453.514,Z 293.995,A -85,B 0,C 180,E1 -8257.746,E2 -8257.746} C_VEL
LIN {X 0,Y 453.525,Z 293.996,A -85,B 0,C 180,E1 -8261.008,E2 -8261.008} C_VEL
LIN {X 0,Y 453.571,Z 293.989,A -85,B 0,C 180,E1 -8263.88,E2 -8263.88} C_VEL
LIN {X 0,Y 453.566,Z 293.991,A -85,B 0,C 180,E1 -8267.471,E2 -8267.471} C_VEL
LIN {X 0,Y 453.592,Z 293.983,A -85,B 0,C 180,E1 -8271.086,E2 -8271.086} C_VEL
LIN {X 0,Y 453.67,Z 293.976,A -85,B 0,C 180,E1 -8273.774,E2 -8273.774} C_VEL
LIN {X 0,Y 453.745,Z 293.964,A -85,B 0,C 180,E1 -8277.336,E2 -8277.336} C_VEL
LIN {X 0,Y 453.824,Z 293.956,A -85,B 0,C 180,E1 -8280,E2 -8280} C_VEL
LIN {X 0,Y 453.746,Z 293.961,A -85,B 0,C 180,E1 -8282.663,E2 -8282.663} C_VEL
LIN {X 0,Y 453.652,Z 293.975,A -85,B 0,C 180,E1 -8286.225,E2 -8286.225} C_VEL
LIN {X 0,Y 453.592,Z 293.98,A -85,B 0,C 180,E1 -8288.913,E2 -8288.913} C_VEL
LIN {X 0,Y 453.565,Z 293.986,A -85,B 0,C 180,E1 -8292.529,E2 -8292.529} C_VEL
LIN {X 0,Y 453.546,Z 293.991,A -85,B 0,C 180,E1 -8296.196,E2 -8296.196} C_VEL
LIN {X 0,Y 453.518,Z 293.991,A -85,B 0,C 180,E1 -8299.039,E2 -8299.039} C_VEL
LIN {X 0,Y 453.478,Z 293.992,A -85,B 0,C 180,E1 -8301.836,E2 -8301.836} C_VEL
LIN {X 0,Y 453.515,Z 293.991,A -85,B 0,C 180,E1 -8304.734,E2 -8304.734} C_VEL
LIN {X 0,Y 453.534,Z 293.983,A -85,B 0,C 180,E1 -8307.959,E2 -8307.959} C_VEL
LIN {X 0,Y 453.467,Z 293.995,A -85,B 0,C 180,E1 -8311.525,E2 -8311.525} C_VEL
LIN {X 0,Y 453.484,Z 293.996,A -85,B 0,C 180,E1 -8314.776,E2 -8314.776} C_VEL
LIN {X 0,Y 453.465,Z 293.994,A -85,B 0,C 180,E1 -8318.312,E2 -8318.312} C_VEL
LIN {X 0,Y 453.495,Z 293.992,A -85,B 0,C 180,E1 -8320.609,E2 -8320.609} C_VEL
LIN {X 0,Y 453.457,Z 294.002,A -85,B 0,C 180,E1 -8323.244,E2 -8323.244} C_VEL
LIN {X 0,Y 453.465,Z 293.999,A -85,B 0,C 180,E1 -8325.779,E2 -8325.779} C_VEL
LIN {X 0,Y 453.481,Z 293.994,A -85,B 0,C 180,E1 -8328.209,E2 -8328.209} C_VEL
LIN {X 0,Y 453.489,Z 293.994,A -85,B 0,C 180,E1 -8330.794,E2 -8330.794} C_VEL
LIN {X 0,Y 453.457,Z 294.006,A -85,B 0,C 180,E1 -8333.917,E2 -8333.917} C_VEL
LIN {X 0,Y 453.485,Z 294,A -85,B 0,C 180,E1 -8337.151,E2 -8337.151} C_VEL
LIN {X 0,Y 453.477,Z 293.999,A -85,B 0,C 180,E1 -8340.268,E2 -8340.268} C_VEL
LIN {X 0,Y 453.518,Z 293.997,A -85,B 0,C 180,E1 -8343.294,E2 -8343.294} C_VEL
LIN {X 0,Y 453.579,Z 294.174,A -85,B 0,C 180,E1 -8343.836,E2 -8343.836} C_VEL
LIN {X 0,Y 455.685,Z 305.35,A -85,B 0,C 180,E1 -8345.949,E2 -8345.949} C_VEL
LIN {X 0,Y 455.356,Z 316.797,A -85,B 0,C 180,E1 -8347.955,E2 -8347.955} C_VEL
LIN {X 0,Y 454.671,Z 334.714,A -85,B 0,C 180,E1 -8351.058,E2 -8351.058} C_VEL
LIN {X 0,Y 454.362,Z 342.373,A -85,B 0,C 180,E1 -8352.372,E2 -8352.372} C_VEL
LIN {X 0,Y 457.612,Z 364.665,A -85,B 0,C 180,E1 -8352.895,E2 -8352.895} C_VEL
LIN {X 0,Y 456.737,Z 451.482,A -85,B 0,C 180,E1 -8354.35,E2 -8354.35} C_VEL
LIN {X 0,Y 456.333,Z 464.528,A -85,B 0,C 180,E1 -8354.736,E2 -8354.736} C_VEL
LIN {X 0,Y 455.786,Z 477.746,A -85,B 0,C 180,E1 -8355.317,E2 -8355.317} C_VEL
LIN {X 0,Y 455.213,Z 489.696,A -85,B 0,C 180,E1 -8356.04,E2 -8356.04} C_VEL
LIN {X 0,Y 454.704,Z 501.244,A -85,B 0,C 180,E1 -8356.939,E2 -8356.939} C_VEL
LIN {X 0,Y 454.207,Z 511.597,A -85,B 0,C 180,E1 -8357.942,E2 -8357.942} C_VEL
LIN {X 0,Y 453.634,Z 520.926,A -85,B 0,C 180,E1 -8359.059,E2 -8359.059} C_VEL
LIN {X 0,Y 453.177,Z 530.004,A -85,B 0,C 180,E1 -8360.403,E2 -8360.403} C_VEL
LIN {X 0,Y 452.902,Z 537.323,A -85,B 0,C 180,E1 -8361.747,E2 -8361.747} C_VEL
LIN {X 0,Y 452.688,Z 542.261,A -85,B 0,C 180,E1 -8362.865,E2 -8362.865} C_VEL
LIN {X 0,Y 452.556,Z 547.066,A -85,B 0,C 180,E1 -8364.206,E2 -8364.206} C_VEL
LIN {X 0,Y 452.487,Z 550.74,A -85,B 0,C 180,E1 -8365.545,E2 -8365.545} C_VEL
LIN {X 0,Y 452.482,Z 552.637,A -85,B 0,C 180,E1 -8366.438,E2 -8366.438} C_VEL
LIN {X 0,Y 452.508,Z 554.061,A -85,B 0,C 180,E1 -8367.329,E2 -8367.329} C_VEL
LIN {X 0,Y 452.457,Z 555.702,A -85,B 0,C 180,E1 -8369.109,E2 -8369.109} C_VEL
LIN {X 0,Y 452.465,Z 555.923,A -85,B 0,C 180,E1 -8369.999,E2 -8369.999} C_VEL
LIN {X 0,Y 452.457,Z 555.703,A -85,B 0,C 180,E1 -8370.889,E2 -8370.889} C_VEL
LIN {X 0,Y 452.507,Z 554.082,A -85,B 0,C 180,E1 -8372.67,E2 -8372.67} C_VEL
LIN {X 0,Y 452.483,Z 552.653,A -85,B 0,C 180,E1 -8373.561,E2 -8373.561} C_VEL
LIN {X 0,Y 452.544,Z 549.67,A -85,B 0,C 180,E1 -8374.899,E2 -8374.899} C_VEL
LIN {X 0,Y 452.61,Z 545.061,A -85,B 0,C 180,E1 -8376.395,E2 -8376.395} C_VEL
LIN {X 0,Y 452.8,Z 539.384,A -85,B 0,C 180,E1 -8377.805,E2 -8377.805} C_VEL
LIN {X 0,Y 453.062,Z 532.58,A -85,B 0,C 180,E1 -8379.148,E2 -8379.148} C_VEL
LIN {X 0,Y 453.457,Z 524.123,A -85,B 0,C 180,E1 -8380.492,E2 -8380.492} C_VEL
LIN {X 0,Y 453.965,Z 515.405,A -85,B 0,C 180,E1 -8381.61,E2 -8381.61} C_VEL
LIN {X 0,Y 454.514,Z 504.184,A -85,B 0,C 180,E1 -8382.775,E2 -8382.775} C_VEL
LIN {X 0,Y 454.976,Z 493.997,A -85,B 0,C 180,E1 -8383.624,E2 -8383.624} C_VEL
LIN {X 0,Y 455.526,Z 482.088,A -85,B 0,C 180,E1 -8384.405,E2 -8384.405} C_VEL
LIN {X 0,Y 456.077,Z 469.732,A -85,B 0,C 180,E1 -8385.015,E2 -8385.015} C_VEL
LIN {X 0,Y 456.474,Z 457.096,A -85,B 0,C 180,E1 -8385.458,E2 -8385.458} C_VEL
LIN {X 0,Y 456.755,Z 442.306,A -85,B 0,C 180,E1 -8385.763,E2 -8385.763} C_VEL
LIN {X 0,Y 457.432,Z 363.659,A -85,B 0,C 180,E1 -8387.052,E2 -8387.052} C_VEL
LIN {X 0,Y 454.338,Z 343.29,A -85,B 0,C 180,E1 -8387.535,E2 -8387.535} C_VEL
LIN {X 0,Y 455.099,Z 327.621,A -85,B 0,C 180,E1 -8390.331,E2 -8390.331} C_VEL
LIN {X 0,Y 456.044,Z 309.418,A -85,B 0,C 180,E1 -8393.62,E2 -8393.62} C_VEL
LIN {X 0,Y 455.594,Z 304.19,A -85,B 0,C 180,E1 -8394.613,E2 -8394.613} C_VEL
LIN {X 0,Y 453.558,Z 293.989,A -85,B 0,C 180,E1 -8396.66,E2 -8396.66} C_VEL
LIN {X 0,Y 453.471,Z 294.001,A -85,B 0,C 180,E1 -8399.784,E2 -8399.784} C_VEL
LIN {X 0,Y 453.488,Z 293.991,A -85,B 0,C 180,E1 -8403.189,E2 -8403.189} C_VEL
LIN {X 0,Y 453.451,Z 294.004,A -85,B 0,C 180,E1 -8406.298,E2 -8406.298} C_VEL
LIN {X 0,Y 453.48,Z 293.992,A -85,B 0,C 180,E1 -8409.45,E2 -8409.45} C_VEL
LIN {X 0,Y 453.473,Z 293.996,A -85,B 0,C 180,E1 -8411.934,E2 -8411.934} C_VEL
LIN {X 0,Y 453.488,Z 293.991,A -85,B 0,C 180,E1 -8415.47,E2 -8415.47} C_VEL
LIN {X 0,Y 453.478,Z 293.996,A -85,B 0,C 180,E1 -8418.209,E2 -8418.209} C_VEL
LIN {X 0,Y 453.511,Z 293.995,A -85,B 0,C 180,E1 -8420.789,E2 -8420.789} C_VEL
LIN {X 0,Y 453.452,Z 293.996,A -85,B 0,C 180,E1 -8423.917,E2 -8423.917} C_VEL
LIN {X 0,Y 453.478,Z 293.997,A -85,B 0,C 180,E1 -8427.151,E2 -8427.151} C_VEL
LIN {X 0,Y 453.47,Z 293.995,A -85,B 0,C 180,E1 -8430.268,E2 -8430.268} C_VEL
LIN {X 0,Y 453.501,Z 293.994,A -85,B 0,C 180,E1 -8433.294,E2 -8433.294} C_VEL
LIN {X 0,Y 453.498,Z 293.99,A -85,B 0,C 180,E1 -8436.239,E2 -8436.239} C_VEL
LIN {X 0,Y 453.477,Z 294.001,A -85,B 0,C 180,E1 -8439.117,E2 -8439.117} C_VEL
LIN {X 0,Y 453.505,Z 293.99,A -85,B 0,C 180,E1 -8441.944,E2 -8441.944} C_VEL
LIN {X 0,Y 453.535,Z 293.987,A -85,B 0,C 180,E1 -8444.726,E2 -8444.726} C_VEL
LIN {X 0,Y 453.554,Z 293.983,A -85,B 0,C 180,E1 -8448.379,E2 -8448.379} C_VEL
LIN {X 0,Y 453.646,Z 293.974,A -85,B 0,C 180,E1 -8451.985,E2 -8451.985} C_VEL
LIN {X 0,Y 453.664,Z 293.969,A -85,B 0,C 180,E1 -8454.667,E2 -8454.667} C_VEL
LIN {X 0,Y 453.738,Z 293.964,A -85,B 0,C 180,E1 -8457.337,E2 -8457.337} C_VEL
LIN {X 0,Y 453.816,Z 293.955,A -85,B 0,C 180,E1 -8460,E2 -8460} C_VEL
LIN {X 0,Y 453.739,Z 293.96,A -85,B 0,C 180,E1 -8462.664,E2 -8462.664} C_VEL
LIN {X 0,Y 453.646,Z 293.976,A -85,B 0,C 180,E1 -8466.226,E2 -8466.226} C_VEL
LIN {X 0,Y 453.586,Z 293.979,A -85,B 0,C 180,E1 -8468.914,E2 -8468.914} C_VEL
LIN {X 0,Y 453.558,Z 293.985,A -85,B 0,C 180,E1 -8472.529,E2 -8472.529} C_VEL
LIN {X 0,Y 453.539,Z 293.993,A -85,B 0,C 180,E1 -8476.196,E2 -8476.196} C_VEL
LIN {X 0,Y 453.512,Z 293.989,A -85,B 0,C 180,E1 -8479.04,E2 -8479.04} C_VEL
LIN {X 0,Y 453.471,Z 293.996,A -85,B 0,C 180,E1 -8481.837,E2 -8481.837} C_VEL
LIN {X 0,Y 453.495,Z 293.994,A -85,B 0,C 180,E1 -8484.736,E2 -8484.736} C_VEL
LIN {X 0,Y 453.502,Z 293.992,A -85,B 0,C 180,E1 -8487.954,E2 -8487.954} C_VEL
LIN {X 0,Y 453.471,Z 293.999,A -85,B 0,C 180,E1 -8490.76,E2 -8490.76} C_VEL
LIN {X 0,Y 453.473,Z 293.994,A -85,B 0,C 180,E1 -8493.914,E2 -8493.914} C_VEL
LIN {X 0,Y 453.449,Z 293.999,A -85,B 0,C 180,E1 -8497.191,E2 -8497.191} C_VEL
LIN {X 0,Y 453.49,Z 293.997,A -85,B 0,C 180,E1 -8500.61,E2 -8500.61} C_VEL
LIN {X 0,Y 453.458,Z 293.996,A -85,B 0,C 180,E1 -8504.223,E2 -8504.223} C_VEL
LIN {X 0,Y 453.436,Z 294.007,A -85,B 0,C 180,E1 -8507.003,E2 -8507.003} C_VEL
LIN {X 0,Y 453.469,Z 293.997,A -85,B 0,C 180,E1 -8509.414,E2 -8509.414} C_VEL
LIN {X 0,Y 453.451,Z 294,A -85,B 0,C 180,E1 -8512.811,E2 -8512.811} C_VEL
LIN {X 0,Y 453.468,Z 293.994,A -85,B 0,C 180,E1 -8516.087,E2 -8516.087} C_VEL
LIN {X 0,Y 453.465,Z 294.002,A -85,B 0,C 180,E1 -8519.241,E2 -8519.241} C_VEL
LIN {X 0,Y 453.475,Z 293.993,A -85,B 0,C 180,E1 -8522.294,E2 -8522.294} C_VEL
LIN {X 0,Y 453.469,Z 293.999,A -85,B 0,C 180,E1 -8525.264,E2 -8525.264} C_VEL
LIN {X 0,Y 453.483,Z 293.992,A -85,B 0,C 180,E1 -8528.416,E2 -8528.416} C_VEL
LIN {X 0,Y 453.525,Z 293.988,A -85,B 0,C 180,E1 -8531.009,E2 -8531.009} C_VEL
LIN {X 0,Y 453.541,Z 293.991,A -85,B 0,C 180,E1 -8533.894,E2 -8533.894} C_VEL
LIN {X 0,Y 453.568,Z 293.985,A -85,B 0,C 180,E1 -8537.472,E2 -8537.472} C_VEL
LIN {X 0,Y 453.559,Z 293.983,A -85,B 0,C 180,E1 -8541.087,E2 -8541.087} C_VEL
LIN {X 0,Y 453.589,Z 293.979,A -85,B 0,C 180,E1 -8543.069,E2 -8543.069} C_VEL
LIN {X 0,Y 452.907,Z 294.071,A -85,B 0,C 180,E1 -8543.81,E2 -8543.81} C_VEL
LIN {X 0,Y 449.953,Z 294.434,A -85,B 0,C 180,E1 -8545.011,E2 -8545.011} C_VEL
LIN {X 0,Y 447.518,Z 294.743,A -85,B 0,C 180,E1 -8545.981,E2 -8545.981} C_VEL
LIN {X 0,Y 446.571,Z 294.854,A -85,B 0,C 180,E1 -8546.732,E2 -8546.732} C_VEL
LIN {X 0,Y 446.547,Z 294.856,A -85,B 0,C 180,E1 -8546.985,E2 -8546.985} C_VEL
LIN {X 0,Y 446.721,Z 294.84,A -85,B 0,C 180,E1 -8550.001,E2 -8550.001} C_VEL
LIN {X 0,Y 446.633,Z 294.848,A -85,B 0,C 180,E1 -8552.706,E2 -8552.706} C_VEL
LIN {X 0,Y 446.609,Z 294.857,A -85,B 0,C 180,E1 -8556.325,E2 -8556.325} C_VEL
LIN {X 0,Y 446.505,Z 294.862,A -85,B 0,C 180,E1 -8559.057,E2 -8559.057} C_VEL
LIN {X 0,Y 446.497,Z 294.868,A -85,B 0,C 180,E1 -8562.731,E2 -8562.731} C_VEL
LIN {X 0,Y 446.463,Z 294.87,A -85,B 0,C 180,E1 -8566.211,E2 -8566.211} C_VEL
LIN {X 0,Y 446.437,Z 294.872,A -85,B 0,C 180,E1 -8569.305,E2 -8569.305} C_VEL
LIN {X 0,Y 446.413,Z 294.877,A -85,B 0,C 180,E1 -8572.2,E2 -8572.2} C_VEL
LIN {X 0,Y 446.469,Z 294.998,A -85,B 0,C 180,E1 -8575.557,E2 -8575.557} C_VEL
LIN {X 0,Y 447.815,Z 302.661,A -85,B 0,C 180,E1 -8577.326,E2 -8577.326} C_VEL
LIN {X 0,Y 447.561,Z 311.726,A -85,B 0,C 180,E1 -8579.291,E2 -8579.291} C_VEL
LIN {X 0,Y 450.873,Z 329.217,A -85,B 0,C 180,E1 -8579.728,E2 -8579.728} C_VEL
LIN {X 0,Y 449.872,Z 419.749,A -85,B 0,C 180,E1 -8581.262,E2 -8581.262} C_VEL
LIN {X 0,Y 449.492,Z 433.33,A -85,B 0,C 180,E1 -8581.686,E2 -8581.686} C_VEL
LIN {X 0,Y 449.154,Z 445.205,A -85,B 0,C 180,E1 -8582.232,E2 -8582.232} C_VEL
LIN {X 0,Y 448.545,Z 457.768,A -85,B 0,C 180,E1 -8583.012,E2 -8583.012} C_VEL
LIN {X 0,Y 447.984,Z 469.417,A -85,B 0,C 180,E1 -8583.949,E2 -8583.949} C_VEL
LIN {X 0,Y 447.513,Z 479.542,A -85,B 0,C 180,E1 -8584.975,E2 -8584.975} C_VEL
LIN {X 0,Y 446.972,Z 488.808,A -85,B 0,C 180,E1 -8586.131,E2 -8586.131} C_VEL
LIN {X 0,Y 446.502,Z 496.508,A -85,B 0,C 180,E1 -8587.301,E2 -8587.301} C_VEL
LIN {X 0,Y 446.08,Z 504.484,A -85,B 0,C 180,E1 -8588.8,E2 -8588.8} C_VEL
LIN {X 0,Y 445.811,Z 510.552,A -85,B 0,C 180,E1 -8590.267,E2 -8590.267} C_VEL
LIN {X 0,Y 445.633,Z 514.547,A -85,B 0,C 180,E1 -8591.482,E2 -8591.482} C_VEL
LIN {X 0,Y 445.525,Z 517.698,A -85,B 0,C 180,E1 -8592.712,E2 -8592.712} C_VEL
LIN {X 0,Y 445.386,Z 520.051,A -85,B 0,C 180,E1 -8593.972,E2 -8593.972} C_VEL
LIN {X 0,Y 445.301,Z 521.621,A -85,B 0,C 180,E1 -8595.253,E2 -8595.253} C_VEL
LIN {X 0,Y 445.243,Z 522.397,A -85,B 0,C 180,E1 -8596.56,E2 -8596.56} C_VEL
LIN {X 0,Y 445.283,Z 522.336,A -85,B 0,C 180,E1 -8597.886,E2 -8597.886} C_VEL
LIN {X 0,Y 445.308,Z 520.85,A -85,B 0,C 180,E1 -8599.678,E2 -8599.678} C_VEL
LIN {X 0,Y 445.428,Z 518.991,A -85,B 0,C 180,E1 -8600.866,E2 -8600.866} C_VEL
LIN {X 0,Y 445.599,Z 516.401,A -85,B 0,C 180,E1 -8602.055,E2 -8602.055} C_VEL
LIN {X 0,Y 445.805,Z 512.102,A -85,B 0,C 180,E1 -8603.514,E2 -8603.514} C_VEL
LIN {X 0,Y 446.107,Z 506.314,A -85,B 0,C 180,E1 -8605.006,E2 -8605.006} C_VEL
LIN {X 0,Y 446.483,Z 498.719,A -85,B 0,C 180,E1 -8606.539,E2 -8606.539} C_VEL
LIN {X 0,Y 446.931,Z 491.679,A -85,B 0,C 180,E1 -8607.679,E2 -8607.679} C_VEL
LIN {X 0,Y 447.495,Z 482.448,A -85,B 0,C 180,E1 -8608.902,E2 -8608.902} C_VEL
LIN {X 0,Y 448.042,Z 472.21,A -85,B 0,C 180,E1 -8610,E2 -8610} C_VEL
LIN {X 0,Y 448.63,Z 461.222,A -85,B 0,C 180,E1 -8610.946,E2 -8610.946} C_VEL
LIN {X 0,Y 449.108,Z 449.885,A -85,B 0,C 180,E1 -8611.712,E2 -8611.712} C_VEL
LIN {X 0,Y 449.583,Z 437.931,A -85,B 0,C 180,E1 -8612.326,E2 -8612.326} C_VEL
LIN {X 0,Y 449.919,Z 424.848,A -85,B 0,C 180,E1 -8612.806,E2 -8612.806} C_VEL
LIN {X 0,Y 450.207,Z 410.544,A -85,B 0,C 180,E1 -8613.113,E2 -8613.113} C_VEL
LIN {X 0,Y 451.117,Z 328.069,A -85,B 0,C 180,E1 -8614.508,E2 -8614.508} C_VEL
LIN {X 0,Y 447.719,Z 311.207,A -85,B 0,C 180,E1 -8614.97,E2 -8614.97} C_VEL
LIN {X 0,Y 447.835,Z 301.814,A -85,B 0,C 180,E1 -8616.655,E2 -8616.655} C_VEL
LIN {X 0,Y 446.464,Z 294.872,A -85,B 0,C 180,E1 -8618.009,E2 -8618.009} C_VEL
LIN {X 0,Y 446.476,Z 294.872,A -85,B 0,C 180,E1 -8620.815,E2 -8620.815} C_VEL
LIN {X 0,Y 446.511,Z 294.867,A -85,B 0,C 180,E1 -8624.48,E2 -8624.48} C_VEL
LIN {X 0,Y 446.519,Z 294.863,A -85,B 0,C 180,E1 -8628.193,E2 -8628.193} C_VEL
LIN {X 0,Y 446.602,Z 294.856,A -85,B 0,C 180,E1 -8631.858,E2 -8631.858} C_VEL
LIN {X 0,Y 446.642,Z 294.847,A -85,B 0,C 180,E1 -8634.582,E2 -8634.582} C_VEL
LIN {X 0,Y 446.665,Z 294.846,A -85,B 0,C 180,E1 -8638.196,E2 -8638.196} C_VEL
LIN {X 0,Y 446.794,Z 294.832,A -85,B 0,C 180,E1 -8640,E2 -8640} C_VEL
LIN {X 0,Y 446.693,Z 294.84,A -85,B 0,C 180,E1 -8642.705,E2 -8642.705} C_VEL
LIN {X 0,Y 446.62,Z 294.85,A -85,B 0,C 180,E1 -8646.324,E2 -8646.324} C_VEL
LIN {X 0,Y 446.538,Z 294.858,A -85,B 0,C 180,E1 -8649.055,E2 -8649.055} C_VEL
LIN {X 0,Y 446.524,Z 294.86,A -85,B 0,C 180,E1 -8652.73,E2 -8652.73} C_VEL
LIN {X 0,Y 446.497,Z 294.869,A -85,B 0,C 180,E1 -8656.227,E2 -8656.227} C_VEL
LIN {X 0,Y 446.47,Z 294.867,A -85,B 0,C 180,E1 -8659.303,E2 -8659.303} C_VEL
LIN {X 0,Y 446.42,Z 294.874,A -85,B 0,C 180,E1 -8662.199,E2 -8662.199} C_VEL
LIN {X 0,Y 446.459,Z 294.87,A -85,B 0,C 180,E1 -8665.152,E2 -8665.152} C_VEL
LIN {X 0,Y 446.486,Z 294.861,A -85,B 0,C 180,E1 -8668.178,E2 -8668.178} C_VEL
LIN {X 0,Y 446.42,Z 294.871,A -85,B 0,C 180,E1 -8671.775,E2 -8671.775} C_VEL
LIN {X 0,Y 446.424,Z 294.874,A -85,B 0,C 180,E1 -8674.523,E2 -8674.523} C_VEL
LIN {X 0,Y 446.416,Z 294.872,A -85,B 0,C 180,E1 -8678.079,E2 -8678.079} C_VEL
LIN {X 0,Y 446.429,Z 294.875,A -85,B 0,C 180,E1 -8680.917,E2 -8680.917} C_VEL
LIN {X 0,Y 446.402,Z 294.879,A -85,B 0,C 180,E1 -8683.846,E2 -8683.846} C_VEL
LIN {X 0,Y 446.4,Z 294.876,A -85,B 0,C 180,E1 -8686.403,E2 -8686.403} C_VEL
LIN {X 0,Y 446.428,Z 294.875,A -85,B 0,C 180,E1 -8689.082,E2 -8689.082} C_VEL
LIN {X 0,Y 446.41,Z 294.88,A -85,B 0,C 180,E1 -8692.121,E2 -8692.121} C_VEL
LIN {X 0,Y 446.432,Z 294.88,A -85,B 0,C 180,E1 -8695.477,E2 -8695.477} C_VEL
LIN {X 0,Y 446.418,Z 294.877,A -85,B 0,C 180,E1 -8698.699,E2 -8698.699} C_VEL
LIN {X 0,Y 446.487,Z 294.871,A -85,B 0,C 180,E1 -8701.821,E2 -8701.821} C_VEL
LIN {X 0,Y 446.523,Z 295.002,A -85,B 0,C 180,E1 -8703.59,E2 -8703.59} C_VEL
LIN {X 0,Y 448.697,Z 306.283,A -85,B 0,C 180,E1 -8705.76,E2 -8705.76} C_VEL
LIN {X 0,Y 448.684,Z 312.88,A -85,B 0,C 180,E1 -8706.946,E2 -8706.946} C_VEL
LIN {X 0,Y 447.834,Z 332.046,A -85,B 0,C 180,E1 -8710.322,E2 -8710.322} C_VEL
LIN {X 0,Y 447.398,Z 342.196,A -85,B 0,C 180,E1 -8712.076,E2 -8712.076} C_VEL
LIN {X 0,Y 450.848,Z 365.142,A -85,B 0,C 180,E1 -8712.63,E2 -8712.63} C_VEL
LIN {X 0,Y 449.918,Z 451.557,A -85,B 0,C 180,E1 -8714.106,E2 -8714.106} C_VEL
LIN {X 0,Y 449.498,Z 464.478,A -85,B 0,C 180,E1 -8714.498,E2 -8714.498} C_VEL
LIN {X 0,Y 448.93,Z 477.623,A -85,B 0,C 180,E1 -8715.088,E2 -8715.088} C_VEL
LIN {X 0,Y 448.329,Z 489.53,A -85,B 0,C 180,E1 -8715.821,E2 -8715.821} C_VEL
LIN {X 0,Y 447.796,Z 500.359,A -85,B 0,C 180,E1 -8716.673,E2 -8716.673} C_VEL
LIN {X 0,Y 447.233,Z 511.367,A -85,B 0,C 180,E1 -8717.752,E2 -8717.752} C_VEL
LIN {X 0,Y 446.642,Z 520.679,A -85,B 0,C 180,E1 -8718.886,E2 -8718.886} C_VEL
LIN {X 0,Y 446.157,Z 529.747,A -85,B 0,C 180,E1 -8720.25,E2 -8720.25} C_VEL
LIN {X 0,Y 445.837,Z 537.065,A -85,B 0,C 180,E1 -8721.615,E2 -8721.615} C_VEL
LIN {X 0,Y 445.616,Z 542.005,A -85,B 0,C 180,E1 -8722.751,E2 -8722.751} C_VEL
LIN {X 0,Y 445.481,Z 546.253,A -85,B 0,C 180,E1 -8723.94,E2 -8723.94} C_VEL
LIN {X 0,Y 445.412,Z 550.485,A -85,B 0,C 180,E1 -8725.475,E2 -8725.475} C_VEL
LIN {X 0,Y 445.381,Z 552.379,A -85,B 0,C 180,E1 -8726.381,E2 -8726.381} C_VEL
LIN {X 0,Y 445.433,Z 553.803,A -85,B 0,C 180,E1 -8727.286,E2 -8727.286} C_VEL
LIN {X 0,Y 445.365,Z 555.441,A -85,B 0,C 180,E1 -8729.095,E2 -8729.095} C_VEL
LIN {X 0,Y 445.371,Z 555.657,A -85,B 0,C 180,E1 -8729.999,E2 -8729.999} C_VEL
LIN {X 0,Y 445.365,Z 555.433,A -85,B 0,C 180,E1 -8730.904,E2 -8730.904} C_VEL
LIN {X 0,Y 445.432,Z 553.806,A -85,B 0,C 180,E1 -8732.712,E2 -8732.712} C_VEL
LIN {X 0,Y 445.382,Z 552.367,A -85,B 0,C 180,E1 -8733.618,E2 -8733.618} C_VEL
LIN {X 0,Y 445.473,Z 549.376,A -85,B 0,C 180,E1 -8734.977,E2 -8734.977} C_VEL
LIN {X 0,Y 445.529,Z 545.154,A -85,B 0,C 180,E1 -8736.385,E2 -8736.385} C_VEL
LIN {X 0,Y 445.727,Z 539.059,A -85,B 0,C 180,E1 -8737.93,E2 -8737.93} C_VEL
LIN {X 0,Y 446.025,Z 532.237,A -85,B 0,C 180,E1 -8739.294,E2 -8739.294} C_VEL
LIN {X 0,Y 446.446,Z 523.753,A -85,B 0,C 180,E1 -8740.659,E2 -8740.659} C_VEL
LIN {X 0,Y 446.974,Z 515.008,A -85,B 0,C 180,E1 -8741.794,E2 -8741.794} C_VEL
LIN {X 0,Y 447.513,Z 504.66,A -85,B 0,C 180,E1 -8742.89,E2 -8742.89} C_VEL
LIN {X 0,Y 448.045,Z 493.527,A -85,B 0,C 180,E1 -8743.839,E2 -8743.839} C_VEL
LIN {X 0,Y 448.621,Z 481.541,A -85,B 0,C 180,E1 -8744.631,E2 -8744.631} C_VEL
LIN {X 0,Y 449.207,Z 469.102,A -85,B 0,C 180,E1 -8745.25,E2 -8745.25} C_VEL
LIN {X 0,Y 449.639,Z 456.276,A -85,B 0,C 180,E1 -8745.699,E2 -8745.699} C_VEL
LIN {X 0,Y 449.919,Z 441.094,A -85,B 0,C 180,E1 -8746.009,E2 -8746.009} C_VEL
LIN {X 0,Y 450.578,Z 364.061,A -85,B 0,C 180,E1 -8747.297,E2 -8747.297} C_VEL
LIN {X 0,Y 447.362,Z 343.13,A -85,B 0,C 180,E1 -8747.791,E2 -8747.791} C_VEL
LIN {X 0,Y 448.16,Z 327.301,A -85,B 0,C 180,E1 -8750.661,E2 -8750.661} C_VEL
LIN {X 0,Y 449.112,Z 310.424,A -85,B 0,C 180,E1 -8753.762,E2 -8753.762} C_VEL
LIN {X 0,Y 448.662,Z 305.583,A -85,B 0,C 180,E1 -8754.696,E2 -8754.696} C_VEL
LIN {X 0,Y 446.522,Z 294.865,A -85,B 0,C 180,E1 -8756.867,E2 -8756.867} C_VEL
LIN {X 0,Y 446.426,Z 294.877,A -85,B 0,C 180,E1 -8760.249,E2 -8760.249} C_VEL
LIN {X 0,Y 446.443,Z 294.87,A -85,B 0,C 180,E1 -8763.453,E2 -8763.453} C_VEL
LIN {X 0,Y 446.399,Z 294.877,A -85,B 0,C 180,E1 -8766.745,E2 -8766.745} C_VEL
LIN {X 0,Y 446.438,Z 294.876,A -85,B 0,C 180,E1 -8770.197,E2 -8770.197} C_VEL
LIN {X 0,Y 446.426,Z 294.877,A -85,B 0,C 180,E1 -8772.604,E2 -8772.604} C_VEL
LIN {X 0,Y 446.452,Z 294.869,A -85,B 0,C 180,E1 -8775.103,E2 -8775.103} C_VEL
LIN {X 0,Y 446.426,Z 294.88,A -85,B 0,C 180,E1 -8778.609,E2 -8778.609} C_VEL
LIN {X 0,Y 446.457,Z 294.871,A -85,B 0,C 180,E1 -8780.974,E2 -8780.974} C_VEL
LIN {X 0,Y 446.416,Z 294.876,A -85,B 0,C 180,E1 -8784.374,E2 -8784.374} C_VEL
LIN {X 0,Y 446.417,Z 294.872,A -85,B 0,C 180,E1 -8787.638,E2 -8787.638} C_VEL
LIN {X 0,Y 446.443,Z 294.876,A -85,B 0,C 180,E1 -8790.79,E2 -8790.79} C_VEL
LIN {X 0,Y 446.472,Z 294.866,A -85,B 0,C 180,E1 -8793.848,E2 -8793.848} C_VEL
LIN {X 0,Y 446.424,Z 294.876,A -85,B 0,C 180,E1 -8796.823,E2 -8796.823} C_VEL
LIN {X 0,Y 446.438,Z 294.871,A -85,B 0,C 180,E1 -8799.737,E2 -8799.737} C_VEL
LIN {X 0,Y 446.457,Z 294.868,A -85,B 0,C 180,E1 -8802.597,E2 -8802.597} C_VEL
LIN {X 0,Y 446.466,Z 294.873,A -85,B 0,C 180,E1 -8805.412,E2 -8805.412} C_VEL
LIN {X 0,Y 446.512,Z 294.861,A -85,B 0,C 180,E1 -8808.193,E2 -8808.193} C_VEL
LIN {X 0,Y 446.594,Z 294.854,A -85,B 0,C 180,E1 -8811.858,E2 -8811.858} C_VEL
LIN {X 0,Y 446.639,Z 294.845,A -85,B 0,C 180,E1 -8814.583,E2 -8814.583} C_VEL
LIN {X 0,Y 446.657,Z 294.844,A -85,B 0,C 180,E1 -8818.197,E2 -8818.197} C_VEL
LIN {X 0,Y 446.786,Z 294.831,A -85,B 0,C 180,E1 -8820,E2 -8820} C_VEL
LIN {X 0,Y 446.686,Z 294.839,A -85,B 0,C 180,E1 -8822.706,E2 -8822.706} C_VEL
LIN {X 0,Y 446.614,Z 294.851,A -85,B 0,C 180,E1 -8826.324,E2 -8826.324} C_VEL
LIN {X 0,Y 446.532,Z 294.858,A -85,B 0,C 180,E1 -8829.056,E2 -8829.056} C_VEL
LIN {X 0,Y 446.516,Z 294.861,A -85,B 0,C 180,E1 -8832.73,E2 -8832.73} C_VEL
LIN {X 0,Y 446.49,Z 294.871,A -85,B 0,C 180,E1 -8836.228,E2 -8836.228} C_VEL
LIN {X 0,Y 446.463,Z 294.866,A -85,B 0,C 180,E1 -8839.304,E2 -8839.304} C_VEL
LIN {X 0,Y 446.413,Z 294.879,A -85,B 0,C 180,E1 -8842.2,E2 -8842.2} C_VEL
LIN {X 0,Y 446.438,Z 294.87,A -85,B 0,C 180,E1 -8845.154,E2 -8845.154} C_VEL
LIN {X 0,Y 446.445,Z 294.873,A -85,B 0,C 180,E1 -8848.182,E2 -8848.182} C_VEL
LIN {X 0,Y 446.411,Z 294.873,A -85,B 0,C 180,E1 -8851.301,E2 -8851.301} C_VEL
LIN {X 0,Y 446.426,Z 294.878,A -85,B 0,C 180,E1 -8854.524,E2 -8854.524} C_VEL
LIN {X 0,Y 446.409,Z 294.874,A -85,B 0,C 180,E1 -8858.079,E2 -8858.079} C_VEL
LIN {X 0,Y 446.416,Z 294.874,A -85,B 0,C 180,E1 -8861.393,E2 -8861.393} C_VEL
LIN {X 0,Y 446.448,Z 294.875,A -85,B 0,C 180,E1 -8865.105,E2 -8865.105} C_VEL
LIN {X 0,Y 446.405,Z 294.876,A -85,B 0,C 180,E1 -8868.607,E2 -8868.607} C_VEL
LIN {X 0,Y 446.41,Z 294.873,A -85,B 0,C 180,E1 -8871.922,E2 -8871.922} C_VEL
LIN {X 0,Y 446.423,Z 294.877,A -85,B 0,C 180,E1 -8875.477,E2 -8875.477} C_VEL
LIN {X 0,Y 446.412,Z 294.874,A -85,B 0,C 180,E1 -8878.7,E2 -8878.7} C_VEL
LIN {X 0,Y 446.425,Z 294.874,A -85,B 0,C 180,E1 -8881.837,E2 -8881.837} C_VEL
LIN {X 0,Y 446.421,Z 294.873,A -85,B 0,C 180,E1 -8884.846,E2 -8884.846} C_VEL
LIN {X 0,Y 446.451,Z 294.869,A -85,B 0,C 180,E1 -8888.246,E2 -8888.246} C_VEL
LIN {X 0,Y 446.45,Z 294.877,A -85,B 0,C 180,E1 -8891.65,E2 -8891.65} C_VEL
LIN {X 0,Y 446.498,Z 294.863,A -85,B 0,C 180,E1 -8894.48,E2 -8894.48} C_VEL
LIN {X 0,Y 446.51,Z 294.864,A -85,B 0,C 180,E1 -8898.193,E2 -8898.193} C_VEL
LIN {X 0,Y 446.51,Z 294.861,A -85,B 0,C 180,E1 -8900.945,E2 -8900.945} C_VEL
LIN {X 0,Y 446.609,Z 294.852,A -85,B 0,C 180,E1 -8903.676,E2 -8903.676} C_VEL
LIN {X 0,Y 446.547,Z 294.856,A -85,B 0,C 180,E1 -8906.985,E2 -8906.985} C_VEL
LIN {X 0,Y 446.332,Z 294.886,A -85,B 0,C 180,E1 -8907.489,E2 -8907.489} C_VEL
LIN {X 0,Y 445.032,Z 295.052,A -85,B 0,C 180,E1 -8908.232,E2 -8908.232} C_VEL
LIN {X 0,Y 440.622,Z 295.599,A -85,B 0,C 180,E1 -8909.947,E2 -8909.947} C_VEL
LIN {X 0,Y 439.572,Z 295.727,A -85,B 0,C 180,E1 -8910.71,E2 -8910.71} C_VEL
LIN {X 0,Y 439.504,Z 295.734,A -85,B 0,C 180,E1 -8910.969,E2 -8910.969} C_VEL
LIN {X 0,Y 439.587,Z 295.725,A -85,B 0,C 180,E1 -8912.75,E2 -8912.75} C_VEL
LIN {X 0,Y 439.599,Z 295.722,A -85,B 0,C 180,E1 -8915.505,E2 -8915.505} C_VEL
LIN {X 0,Y 439.482,Z 295.743,A -85,B 0,C 180,E1 -8918.275,E2 -8918.275} C_VEL
LIN {X 0,Y 439.475,Z 295.739,A -85,B 0,C 180,E1 -8921.999,E2 -8921.999} C_VEL
LIN {X 0,Y 439.381,Z 295.754,A -85,B 0,C 180,E1 -8924.829,E2 -8924.829} C_VEL
LIN {X 0,Y 439.384,Z 295.748,A -85,B 0,C 180,E1 -8927.693,E2 -8927.693} C_VEL
LIN {X 0,Y 439.372,Z 295.756,A -85,B 0,C 180,E1 -8930.604,E2 -8930.604} C_VEL
LIN {X 0,Y 439.35,Z 295.758,A -85,B 0,C 180,E1 -8933.573,E2 -8933.573} C_VEL
LIN {X 0,Y 439.422,Z 295.848,A -85,B 0,C 180,E1 -8935.362,E2 -8935.362} C_VEL
LIN {X 0,Y 440.862,Z 304.036,A -85,B 0,C 180,E1 -8937.279,E2 -8937.279} C_VEL
LIN {X 0,Y 440.633,Z 311.925,A -85,B 0,C 180,E1 -8939.015,E2 -8939.015} C_VEL
LIN {X 0,Y 444.035,Z 329.056,A -85,B 0,C 180,E1 -8939.465,E2 -8939.465} C_VEL
LIN {X 0,Y 443.031,Z 419.364,A -85,B 0,C 180,E1 -8941.019,E2 -8941.019} C_VEL
LIN {X 0,Y 442.589,Z 433.171,A -85,B 0,C 180,E1 -8941.448,E2 -8941.448} C_VEL
LIN {X 0,Y 442.243,Z 445.69,A -85,B 0,C 180,E1 -8942.032,E2 -8942.032} C_VEL
LIN {X 0,Y 441.682,Z 457.205,A -85,B 0,C 180,E1 -8942.752,E2 -8942.752} C_VEL
LIN {X 0,Y 441.131,Z 468.036,A -85,B 0,C 180,E1 -8943.617,E2 -8943.617} C_VEL
LIN {X 0,Y 440.623,Z 478.326,A -85,B 0,C 180,E1 -8944.639,E2 -8944.639} C_VEL
LIN {X 0,Y 440.051,Z 487.967,A -85,B 0,C 180,E1 -8945.822,E2 -8945.822} C_VEL
LIN {X 0,Y 439.498,Z 496.645,A -85,B 0,C 180,E1 -8947.143,E2 -8947.143} C_VEL
LIN {X 0,Y 439.05,Z 504.491,A -85,B 0,C 180,E1 -8948.63,E2 -8948.63} C_VEL
LIN {X 0,Y 438.762,Z 510.71,A -85,B 0,C 180,E1 -8950.145,E2 -8950.145} C_VEL
LIN {X 0,Y 438.537,Z 515.581,A -85,B 0,C 180,E1 -8951.691,E2 -8951.691} C_VEL
LIN {X 0,Y 438.392,Z 518.668,A -85,B 0,C 180,E1 -8953.005,E2 -8953.005} C_VEL
LIN {X 0,Y 438.308,Z 520.124,A -85,B 0,C 180,E1 -8953.817,E2 -8953.817} C_VEL
LIN {X 0,Y 438.222,Z 521.779,A -85,B 0,C 180,E1 -8955.117,E2 -8955.117} C_VEL
LIN {X 0,Y 438.186,Z 522.628,A -85,B 0,C 180,E1 -8956.395,E2 -8956.395} C_VEL
LIN {X 0,Y 438.193,Z 522.673,A -85,B 0,C 180,E1 -8957.652,E2 -8957.652} C_VEL
LIN {X 0,Y 438.208,Z 521.966,A -85,B 0,C 180,E1 -8958.92,E2 -8958.92} C_VEL
LIN {X 0,Y 438.274,Z 520.289,A -85,B 0,C 180,E1 -8960.328,E2 -8960.328} C_VEL
LIN {X 0,Y 438.459,Z 517.57,A -85,B 0,C 180,E1 -8961.759,E2 -8961.759} C_VEL
LIN {X 0,Y 438.664,Z 513.634,A -85,B 0,C 180,E1 -8963.233,E2 -8963.233} C_VEL
LIN {X 0,Y 438.982,Z 508.038,A -85,B 0,C 180,E1 -8964.805,E2 -8964.805} C_VEL
LIN {X 0,Y 439.391,Z 501.247,A -85,B 0,C 180,E1 -8966.278,E2 -8966.278} C_VEL
LIN {X 0,Y 439.901,Z 492.88,A -85,B 0,C 180,E1 -8967.716,E2 -8967.716} C_VEL
LIN {X 0,Y 440.464,Z 484.388,A -85,B 0,C 180,E1 -8968.897,E2 -8968.897} C_VEL
LIN {X 0,Y 440.996,Z 474.691,A -85,B 0,C 180,E1 -8969.999,E2 -8969.999} C_VEL
LIN {X 0,Y 441.641,Z 463.81,A -85,B 0,C 180,E1 -8970.988,E2 -8970.988} C_VEL
LIN {X 0,Y 442.232,Z 451.85,A -85,B 0,C 180,E1 -8971.849,E2 -8971.849} C_VEL
LIN {X 0,Y 442.724,Z 439.336,A -85,B 0,C 180,E1 -8972.525,E2 -8972.525} C_VEL
LIN {X 0,Y 443.078,Z 426.235,A -85,B 0,C 180,E1 -8973.028,E2 -8973.028} C_VEL
LIN {X 0,Y 443.372,Z 413.341,A -85,B 0,C 180,E1 -8973.334,E2 -8973.334} C_VEL
LIN {X 0,Y 444.446,Z 329.216,A -85,B 0,C 180,E1 -8974.785,E2 -8974.785} C_VEL
LIN {X 0,Y 440.853,Z 311.423,A -85,B 0,C 180,E1 -8975.29,E2 -8975.29} C_VEL
LIN {X 0,Y 440.948,Z 303.297,A -85,B 0,C 180,E1 -8976.766,E2 -8976.766} C_VEL
LIN {X 0,Y 439.441,Z 295.746,A -85,B 0,C 180,E1 -8978.238,E2 -8978.238} C_VEL
LIN {X 0,Y 439.427,Z 295.753,A -85,B 0,C 180,E1 -8981.345,E2 -8981.345} C_VEL
LIN {X 0,Y 439.465,Z 295.745,A -85,B 0,C 180,E1 -8984.224,E2 -8984.224} C_VEL
LIN {X 0,Y 439.486,Z 295.741,A -85,B 0,C 180,E1 -8988.001,E2 -8988.001} C_VEL
LIN {X 0,Y 439.55,Z 295.734,A -85,B 0,C 180,E1 -8991.726,E2 -8991.726} C_VEL
LIN {X 0,Y 439.618,Z 295.723,A -85,B 0,C 180,E1 -8994.495,E2 -8994.495} C_VEL
LIN {X 0,Y 439.635,Z 295.721,A -85,B 0,C 180,E1 -8998.168,E2 -8998.168} C_VEL
LIN {X 0,Y 439.764,Z 295.707,A -85,B 0,C 180,E1 -9000,E2 -9000} C_VEL
LIN {X 0,Y 439.642,Z 295.718,A -85,B 0,C 180,E1 -9002.749,E2 -9002.749} C_VEL
LIN {X 0,Y 439.592,Z 295.724,A -85,B 0,C 180,E1 -9006.425,E2 -9006.425} C_VEL
LIN {X 0,Y 439.5,Z 295.734,A -85,B 0,C 180,E1 -9009.201,E2 -9009.201} C_VEL
LIN {X 0,Y 439.468,Z 295.737,A -85,B 0,C 180,E1 -9012.937,E2 -9012.937} C_VEL
LIN {X 0,Y 439.448,Z 295.746,A -85,B 0,C 180,E1 -9016.348,E2 -9016.348} C_VEL
LIN {X 0,Y 439.403,Z 295.747,A -85,B 0,C 180,E1 -9019.626,E2 -9019.626} C_VEL
LIN {X 0,Y 439.366,Z 295.757,A -85,B 0,C 180,E1 -9022.575,E2 -9022.575} C_VEL
LIN {X 0,Y 439.407,Z 295.746,A -85,B 0,C 180,E1 -9025.585,E2 -9025.585} C_VEL
LIN {X 0,Y 439.419,Z 295.745,A -85,B 0,C 180,E1 -9028.673,E2 -9028.673} C_VEL
LIN {X 0,Y 439.37,Z 295.749,A -85,B 0,C 180,E1 -9032.03,E2 -9032.03} C_VEL
LIN {X 0,Y 439.393,Z 295.753,A -85,B 0,C 180,E1 -9035.34,E2 -9035.34} C_VEL
LIN {X 0,Y 439.379,Z 295.75,A -85,B 0,C 180,E1 -9038.595,E2 -9038.595} C_VEL
LIN {X 0,Y 439.39,Z 295.753,A -85,B 0,C 180,E1 -9041.257,E2 -9041.257} C_VEL
LIN {X 0,Y 439.401,Z 295.75,A -85,B 0,C 180,E1 -9044.729,E2 -9044.729} C_VEL
LIN {X 0,Y 439.398,Z 295.751,A -85,B 0,C 180,E1 -9047.796,E2 -9047.796} C_VEL
LIN {X 0,Y 439.397,Z 295.75,A -85,B 0,C 180,E1 -9050.224,E2 -9050.224} C_VEL
LIN {X 0,Y 439.376,Z 295.759,A -85,B 0,C 180,E1 -9053.713,E2 -9053.713} C_VEL
LIN {X 0,Y 439.375,Z 295.758,A -85,B 0,C 180,E1 -9057.054,E2 -9057.054} C_VEL
LIN {X 0,Y 439.385,Z 295.755,A -85,B 0,C 180,E1 -9060.274,E2 -9060.274} C_VEL
LIN {X 0,Y 439.455,Z 295.848,A -85,B 0,C 180,E1 -9063.333,E2 -9063.333} C_VEL
LIN {X 0,Y 441.691,Z 307.184,A -85,B 0,C 180,E1 -9065.562,E2 -9065.562} C_VEL
LIN {X 0,Y 441.876,Z 311.288,A -85,B 0,C 180,E1 -9066.321,E2 -9066.321} C_VEL
LIN {X 0,Y 441.006,Z 330.028,A -85,B 0,C 180,E1 -9069.68,E2 -9069.68} C_VEL
LIN {X 0,Y 440.476,Z 341.733,A -85,B 0,C 180,E1 -9071.753,E2 -9071.753} C_VEL
LIN {X 0,Y 444.078,Z 365.198,A -85,B 0,C 180,E1 -9072.343,E2 -9072.343} C_VEL
LIN {X 0,Y 443.112,Z 451.632,A -85,B 0,C 180,E1 -9073.855,E2 -9073.855} C_VEL
LIN {X 0,Y 442.639,Z 465.179,A -85,B 0,C 180,E1 -9074.281,E2 -9074.281} C_VEL
LIN {X 0,Y 442.079,Z 477.496,A -85,B 0,C 180,E1 -9074.851,E2 -9074.851} C_VEL
LIN {X 0,Y 441.433,Z 489.365,A -85,B 0,C 180,E1 -9075.595,E2 -9075.595} C_VEL
LIN {X 0,Y 440.82,Z 501.065,A -85,B 0,C 180,E1 -9076.538,E2 -9076.538} C_VEL
LIN {X 0,Y 440.263,Z 511.167,A -85,B 0,C 180,E1 -9077.555,E2 -9077.555} C_VEL
LIN {X 0,Y 439.659,Z 520.467,A -85,B 0,C 180,E1 -9078.707,E2 -9078.707} C_VEL
LIN {X 0,Y 439.128,Z 529.527,A -85,B 0,C 180,E1 -9080.093,E2 -9080.093} C_VEL
LIN {X 0,Y 438.784,Z 536.832,A -85,B 0,C 180,E1 -9081.479,E2 -9081.479} C_VEL
LIN {X 0,Y 438.541,Z 541.762,A -85,B 0,C 180,E1 -9082.634,E2 -9082.634} C_VEL
LIN {X 0,Y 438.381,Z 546.445,A -85,B 0,C 180,E1 -9083.982,E2 -9083.982} C_VEL
LIN {X 0,Y 438.341,Z 550.231,A -85,B 0,C 180,E1 -9085.401,E2 -9085.401} C_VEL
LIN {X 0,Y 438.282,Z 552.122,A -85,B 0,C 180,E1 -9086.322,E2 -9086.322} C_VEL
LIN {X 0,Y 438.341,Z 553.544,A -85,B 0,C 180,E1 -9087.243,E2 -9087.243} C_VEL
LIN {X 0,Y 438.295,Z 554.559,A -85,B 0,C 180,E1 -9088.162,E2 -9088.162} C_VEL
LIN {X 0,Y 438.277,Z 555.18,A -85,B 0,C 180,E1 -9089.081,E2 -9089.081} C_VEL
LIN {X 0,Y 438.281,Z 555.391,A -85,B 0,C 180,E1 -9089.999,E2 -9089.999} C_VEL
LIN {X 0,Y 438.277,Z 555.164,A -85,B 0,C 180,E1 -9090.918,E2 -9090.918} C_VEL
LIN {X 0,Y 438.295,Z 554.544,A -85,B 0,C 180,E1 -9091.837,E2 -9091.837} C_VEL
LIN {X 0,Y 438.34,Z 553.529,A -85,B 0,C 180,E1 -9092.756,E2 -9092.756} C_VEL
LIN {X 0,Y 438.283,Z 552.081,A -85,B 0,C 180,E1 -9093.677,E2 -9093.677} C_VEL
LIN {X 0,Y 438.382,Z 549.08,A -85,B 0,C 180,E1 -9095.058,E2 -9095.058} C_VEL
LIN {X 0,Y 438.447,Z 545.007,A -85,B 0,C 180,E1 -9096.442,E2 -9096.442} C_VEL
LIN {X 0,Y 438.671,Z 538.733,A -85,B 0,C 180,E1 -9098.058,E2 -9098.058} C_VEL
LIN {X 0,Y 438.965,Z 531.894,A -85,B 0,C 180,E1 -9099.445,E2 -9099.445} C_VEL
LIN {X 0,Y 439.412,Z 523.38,A -85,B 0,C 180,E1 -9100.831,E2 -9100.831} C_VEL
LIN {X 0,Y 439.974,Z 514.604,A -85,B 0,C 180,E1 -9101.984,E2 -9101.984} C_VEL
LIN {X 0,Y 440.541,Z 504.671,A -85,B 0,C 180,E1 -9103.053,E2 -9103.053} C_VEL
LIN {X 0,Y 441.109,Z 493.018,A -85,B 0,C 180,E1 -9104.061,E2 -9104.061} C_VEL
LIN {X 0,Y 441.733,Z 480.942,A -85,B 0,C 180,E1 -9104.865,E2 -9104.865} C_VEL
LIN {X 0,Y 442.342,Z 468.393,A -85,B 0,C 180,E1 -9105.492,E2 -9105.492} C_VEL
LIN {X 0,Y 442.766,Z 456.326,A -85,B 0,C 180,E1 -9105.92,E2 -9105.92} C_VEL
LIN {X 0,Y 443.07,Z 441.395,A -85,B 0,C 180,E1 -9106.234,E2 -9106.234} C_VEL
LIN {X 0,Y 443.822,Z 365.312,A -85,B 0,C 180,E1 -9107.527,E2 -9107.527} C_VEL
LIN {X 0,Y 440.412,Z 342.794,A -85,B 0,C 180,E1 -9108.081,E2 -9108.081} C_VEL
LIN {X 0,Y 441.263,Z 326.991,A -85,B 0,C 180,E1 -9110.999,E2 -9110.999} C_VEL
LIN {X 0,Y 442.176,Z 311.398,A -85,B 0,C 180,E1 -9113.909,E2 -9113.909} C_VEL
LIN {X 0,Y 441.623,Z 306.416,A -85,B 0,C 180,E1 -9114.892,E2 -9114.892} C_VEL
LIN {X 0,Y 439.487,Z 295.742,A -85,B 0,C 180,E1 -9117.113,E2 -9117.113} C_VEL
LIN {X 0,Y 439.379,Z 295.755,A -85,B 0,C 180,E1 -9120.26,E2 -9120.26} C_VEL
LIN {X 0,Y 439.394,Z 295.75,A -85,B 0,C 180,E1 -9123.723,E2 -9123.723} C_VEL
LIN {X 0,Y 439.345,Z 295.754,A -85,B 0,C 180,E1 -9126.886,E2 -9126.886} C_VEL
LIN {X 0,Y 439.398,Z 295.749,A -85,B 0,C 180,E1 -9129.848,E2 -9129.848} C_VEL
LIN {X 0,Y 439.378,Z 295.755,A -85,B 0,C 180,E1 -9132.626,E2 -9132.626} C_VEL
LIN {X 0,Y 439.402,Z 295.747,A -85,B 0,C 180,E1 -9135.271,E2 -9135.271} C_VEL
LIN {X 0,Y 439.386,Z 295.755,A -85,B 0,C 180,E1 -9138.742,E2 -9138.742} C_VEL
LIN {X 0,Y 439.381,Z 295.749,A -85,B 0,C 180,E1 -9141.605,E2 -9141.605} C_VEL
LIN {X 0,Y 439.396,Z 295.754,A -85,B 0,C 180,E1 -9144.844,E2 -9144.844} C_VEL
LIN {X 0,Y 439.369,Z 295.751,A -85,B 0,C 180,E1 -9148.139,E2 -9148.139} C_VEL
LIN {X 0,Y 439.427,Z 295.744,A -85,B 0,C 180,E1 -9151.598,E2 -9151.598} C_VEL
LIN {X 0,Y 439.4,Z 295.748,A -85,B 0,C 180,E1 -9154.415,E2 -9154.415} C_VEL
LIN {X 0,Y 439.359,Z 295.755,A -85,B 0,C 180,E1 -9157.424,E2 -9157.424} C_VEL
LIN {X 0,Y 439.435,Z 295.744,A -85,B 0,C 180,E1 -9160.663,E2 -9160.663} C_VEL
LIN {X 0,Y 439.457,Z 295.739,A -85,B 0,C 180,E1 -9164.224,E2 -9164.224} C_VEL
LIN {X 0,Y 439.478,Z 295.738,A -85,B 0,C 180,E1 -9168.001,E2 -9168.001} C_VEL
LIN {X 0,Y 439.542,Z 295.734,A -85,B 0,C 180,E1 -9171.726,E2 -9171.726} C_VEL
LIN {X 0,Y 439.614,Z 295.72,A -85,B 0,C 180,E1 -9174.496,E2 -9174.496} C_VEL
LIN {X 0,Y 439.627,Z 295.72,A -85,B 0,C 180,E1 -9178.168,E2 -9178.168} C_VEL
LIN {X 0,Y 439.755,Z 295.707,A -85,B 0,C 180,E1 -9180,E2 -9180} C_VEL
LIN {X 0,Y 439.635,Z 295.717,A -85,B 0,C 180,E1 -9182.749,E2 -9182.749} C_VEL
LIN {X 0,Y 439.586,Z 295.725,A -85,B 0,C 180,E1 -9186.426,E2 -9186.426} C_VEL
LIN {X 0,Y 439.494,Z 295.735,A -85,B 0,C 180,E1 -9189.202,E2 -9189.202} C_VEL
LIN {X 0,Y 439.46,Z 295.739,A -85,B 0,C 180,E1 -9192.938,E2 -9192.938} C_VEL
LIN {X 0,Y 439.441,Z 295.747,A -85,B 0,C 180,E1 -9196.349,E2 -9196.349} C_VEL
LIN {X 0,Y 439.397,Z 295.748,A -85,B 0,C 180,E1 -9199.627,E2 -9199.627} C_VEL
LIN {X 0,Y 439.359,Z 295.757,A -85,B 0,C 180,E1 -9202.576,E2 -9202.576} C_VEL
LIN {X 0,Y 439.375,Z 295.75,A -85,B 0,C 180,E1 -9205.587,E2 -9205.587} C_VEL
LIN {X 0,Y 439.396,Z 295.753,A -85,B 0,C 180,E1 -9208.675,E2 -9208.675} C_VEL
LIN {X 0,Y 439.366,Z 295.752,A -85,B 0,C 180,E1 -9212.031,E2 -9212.031} C_VEL
LIN {X 0,Y 439.391,Z 295.748,A -85,B 0,C 180,E1 -9215.341,E2 -9215.341} C_VEL
LIN {X 0,Y 439.365,Z 295.757,A -85,B 0,C 180,E1 -9218.597,E2 -9218.597} C_VEL
LIN {X 0,Y 439.378,Z 295.752,A -85,B 0,C 180,E1 -9221.256,E2 -9221.256} C_VEL
LIN {X 0,Y 439.396,Z 295.752,A -85,B 0,C 180,E1 -9224.731,E2 -9224.731} C_VEL
LIN {X 0,Y 439.357,Z 295.752,A -85,B 0,C 180,E1 -9227.792,E2 -9227.792} C_VEL
LIN {X 0,Y 439.357,Z 295.752,A -85,B 0,C 180,E1 -9230.221,E2 -9230.221} C_VEL
LIN {X 0,Y 439.372,Z 295.752,A -85,B 0,C 180,E1 -9233.714,E2 -9233.714} C_VEL
LIN {X 0,Y 439.372,Z 295.755,A -85,B 0,C 180,E1 -9237.055,E2 -9237.055} C_VEL
LIN {X 0,Y 439.371,Z 295.75,A -85,B 0,C 180,E1 -9240.274,E2 -9240.274} C_VEL
LIN {X 0,Y 439.365,Z 295.758,A -85,B 0,C 180,E1 -9243.393,E2 -9243.393} C_VEL
LIN {X 0,Y 439.367,Z 295.75,A -85,B 0,C 180,E1 -9246.429,E2 -9246.429} C_VEL
LIN {X 0,Y 439.389,Z 295.753,A -85,B 0,C 180,E1 -9249.398,E2 -9249.398} C_VEL
LIN {X 0,Y 439.402,Z 295.747,A -85,B 0,C 180,E1 -9252.309,E2 -9252.309} C_VEL
LIN {X 0,Y 439.445,Z 295.742,A -85,B 0,C 180,E1 -9255.175,E2 -9255.175} C_VEL
LIN {X 0,Y 439.479,Z 295.743,A -85,B 0,C 180,E1 -9258.002,E2 -9258.002} C_VEL
LIN {X 0,Y 439.483,Z 295.741,A -85,B 0,C 180,E1 -9261.726,E2 -9261.726} C_VEL
LIN {X 0,Y 439.599,Z 295.724,A -85,B 0,C 180,E1 -9264.496,E2 -9264.496} C_VEL
LIN {X 0,Y 439.626,Z 295.726,A -85,B 0,C 180,E1 -9268.168,E2 -9268.168} C_VEL
LIN {X 0,Y 439.672,Z 295.718,A -85,B 0,C 180,E1 -9270.001,E2 -9270.001} C_VEL
LIN {X 0,Y 439.504,Z 295.734,A -85,B 0,C 180,E1 -9270.969,E2 -9270.969} C_VEL
LIN {X 0,Y 438.858,Z 295.818,A -85,B 0,C 180,E1 -9271.734,E2 -9271.734} C_VEL
LIN {X 0,Y 435.92,Z 296.182,A -85,B 0,C 180,E1 -9272.974,E2 -9272.974} C_VEL
LIN {X 0,Y 433.457,Z 296.491,A -85,B 0,C 180,E1 -9273.975,E2 -9273.975} C_VEL
LIN {X 0,Y 432.468,Z 296.613,A -85,B 0,C 180,E1 -9274.75,E2 -9274.75} C_VEL
LIN {X 0,Y 432.426,Z 296.616,A -85,B 0,C 180,E1 -9275.013,E2 -9275.013} C_VEL
LIN {X 0,Y 432.519,Z 296.604,A -85,B 0,C 180,E1 -9277.607,E2 -9277.607} C_VEL
LIN {X 0,Y 432.366,Z 296.623,A -85,B 0,C 180,E1 -9281.249,E2 -9281.249} C_VEL
LIN {X 0,Y 432.389,Z 296.621,A -85,B 0,C 180,E1 -9283.154,E2 -9283.154} C_VEL
LIN {X 0,Y 432.365,Z 296.629,A -85,B 0,C 180,E1 -9286.455,E2 -9286.455} C_VEL
LIN {X 0,Y 432.32,Z 296.629,A -85,B 0,C 180,E1 -9289.962,E2 -9289.962} C_VEL
LIN {X 0,Y 432.302,Z 296.639,A -85,B 0,C 180,E1 -9292.966,E2 -9292.966} C_VEL
LIN {X 0,Y 432.373,Z 296.819,A -85,B 0,C 180,E1 -9295.193,E2 -9295.193} C_VEL
LIN {X 0,Y 433.896,Z 305.302,A -85,B 0,C 180,E1 -9297.205,E2 -9297.205} C_VEL
LIN {X 0,Y 433.699,Z 312.149,A -85,B 0,C 180,E1 -9298.73,E2 -9298.73} C_VEL
LIN {X 0,Y 437.281,Z 330.473,A -85,B 0,C 180,E1 -9299.225,E2 -9299.225} C_VEL
LIN {X 0,Y 436.161,Z 419.726,A -85,B 0,C 180,E1 -9300.787,E2 -9300.787} C_VEL
LIN {X 0,Y 435.723,Z 433.285,A -85,B 0,C 180,E1 -9301.216,E2 -9301.216} C_VEL
LIN {X 0,Y 435.353,Z 446.055,A -85,B 0,C 180,E1 -9301.821,E2 -9301.821} C_VEL
LIN {X 0,Y 434.7,Z 458.961,A -85,B 0,C 180,E1 -9302.657,E2 -9302.657} C_VEL
LIN {X 0,Y 434.122,Z 469.535,A -85,B 0,C 180,E1 -9303.536,E2 -9303.536} C_VEL
LIN {X 0,Y 433.624,Z 479.473,A -85,B 0,C 180,E1 -9304.56,E2 -9304.56} C_VEL
LIN {X 0,Y 433.011,Z 488.861,A -85,B 0,C 180,E1 -9305.754,E2 -9305.754} C_VEL
LIN {X 0,Y 432.491,Z 496.645,A -85,B 0,C 180,E1 -9306.96,E2 -9306.96} C_VEL
LIN {X 0,Y 432.036,Z 504.258,A -85,B 0,C 180,E1 -9308.412,E2 -9308.412} C_VEL
LIN {X 0,Y 431.704,Z 511.059,A -85,B 0,C 180,E1 -9310.079,E2 -9310.079} C_VEL
LIN {X 0,Y 431.477,Z 515.436,A -85,B 0,C 180,E1 -9311.473,E2 -9311.473} C_VEL
LIN {X 0,Y 431.294,Z 519.374,A -85,B 0,C 180,E1 -9313.188,E2 -9313.188} C_VEL
LIN {X 0,Y 431.152,Z 521.387,A -85,B 0,C 180,E1 -9314.501,E2 -9314.501} C_VEL
LIN {X 0,Y 431.101,Z 522.606,A -85,B 0,C 180,E1 -9315.833,E2 -9315.833} C_VEL
LIN {X 0,Y 431.085,Z 523.015,A -85,B 0,C 180,E1 -9317.193,E2 -9317.193} C_VEL
LIN {X 0,Y 431.108,Z 522.548,A -85,B 0,C 180,E1 -9318.582,E2 -9318.582} C_VEL
LIN {X 0,Y 431.15,Z 521.131,A -85,B 0,C 180,E1 -9320.008,E2 -9320.008} C_VEL
LIN {X 0,Y 431.387,Z 518.066,A -85,B 0,C 180,E1 -9321.75,E2 -9321.75} C_VEL
LIN {X 0,Y 431.556,Z 515.104,A -85,B 0,C 180,E1 -9322.946,E2 -9322.946} C_VEL
LIN {X 0,Y 431.84,Z 510.166,A -85,B 0,C 180,E1 -9324.462,E2 -9324.462} C_VEL
LIN {X 0,Y 432.267,Z 503.597,A -85,B 0,C 180,E1 -9326.015,E2 -9326.015} C_VEL
LIN {X 0,Y 432.705,Z 496.745,A -85,B 0,C 180,E1 -9327.313,E2 -9327.313} C_VEL
LIN {X 0,Y 433.242,Z 488.483,A -85,B 0,C 180,E1 -9328.592,E2 -9328.592} C_VEL
LIN {X 0,Y 433.793,Z 480.265,A -85,B 0,C 180,E1 -9329.636,E2 -9329.636} C_VEL
LIN {X 0,Y 434.4,Z 470.031,A -85,B 0,C 180,E1 -9330.703,E2 -9330.703} C_VEL
LIN {X 0,Y 435.107,Z 458.289,A -85,B 0,C 180,E1 -9331.674,E2 -9331.674} C_VEL
LIN {X 0,Y 435.692,Z 446.591,A -85,B 0,C 180,E1 -9332.429,E2 -9332.429} C_VEL
LIN {X 0,Y 436.126,Z 433.457,A -85,B 0,C 180,E1 -9333.052,E2 -9333.052} C_VEL
LIN {X 0,Y 436.49,Z 421.003,A -85,B 0,C 180,E1 -9333.451,E2 -9333.451} C_VEL
LIN {X 0,Y 437.618,Z 341.42,A -85,B 0,C 180,E1 -9334.875,E2 -9334.875} C_VEL
LIN {X 0,Y 437.663,Z 329.63,A -85,B 0,C 180,E1 -9335.091,E2 -9335.091} C_VEL
LIN {X 0,Y 433.953,Z 311.724,A -85,B 0,C 180,E1 -9335.607,E2 -9335.607} C_VEL
LIN {X 0,Y 434.081,Z 304.832,A -85,B 0,C 180,E1 -9336.882,E2 -9336.882} C_VEL
LIN {X 0,Y 432.369,Z 296.629,A -85,B 0,C 180,E1 -9338.547,E2 -9338.547} C_VEL
LIN {X 0,Y 432.387,Z 296.629,A -85,B 0,C 180,E1 -9341.029,E2 -9341.029} C_VEL
LIN {X 0,Y 432.433,Z 296.623,A -85,B 0,C 180,E1 -9343.961,E2 -9343.961} C_VEL
LIN {X 0,Y 432.461,Z 296.617,A -85,B 0,C 180,E1 -9347.803,E2 -9347.803} C_VEL
LIN {X 0,Y 432.494,Z 296.613,A -85,B 0,C 180,E1 -9351.59,E2 -9351.59} C_VEL
LIN {X 0,Y 432.595,Z 296.598,A -85,B 0,C 180,E1 -9354.406,E2 -9354.406} C_VEL
LIN {X 0,Y 432.605,Z 296.597,A -85,B 0,C 180,E1 -9358.138,E2 -9358.138} C_VEL
LIN {X 0,Y 432.734,Z 296.583,A -85,B 0,C 180,E1 -9360,E2 -9360} C_VEL
LIN {X 0,Y 432.594,Z 296.596,A -85,B 0,C 180,E1 -9362.793,E2 -9362.793} C_VEL
LIN {X 0,Y 432.586,Z 296.599,A -85,B 0,C 180,E1 -9365.594,E2 -9365.594} C_VEL
LIN {X 0,Y 432.484,Z 296.614,A -85,B 0,C 180,E1 -9368.41,E2 -9368.41} C_VEL
LIN {X 0,Y 432.461,Z 296.618,A -85,B 0,C 180,E1 -9372.196,E2 -9372.196} C_VEL
LIN {X 0,Y 432.432,Z 296.619,A -85,B 0,C 180,E1 -9376.039,E2 -9376.039} C_VEL
LIN {X 0,Y 432.388,Z 296.621,A -85,B 0,C 180,E1 -9379.485,E2 -9379.485} C_VEL
LIN {X 0,Y 432.32,Z 296.632,A -85,B 0,C 180,E1 -9382.964,E2 -9382.964} C_VEL
LIN {X 0,Y 432.366,Z 296.623,A -85,B 0,C 180,E1 -9386.032,E2 -9386.032} C_VEL
LIN {X 0,Y 432.344,Z 296.63,A -85,B 0,C 180,E1 -9389.187,E2 -9389.187} C_VEL
LIN {X 0,Y 432.324,Z 296.629,A -85,B 0,C 180,E1 -9392.443,E2 -9392.443} C_VEL
LIN {X 0,Y 432.344,Z 296.629,A -85,B 0,C 180,E1 -9395.631,E2 -9395.631} C_VEL
LIN {X 0,Y 432.342,Z 296.627,A -85,B 0,C 180,E1 -9398.714,E2 -9398.714} C_VEL
LIN {X 0,Y 432.335,Z 296.631,A -85,B 0,C 180,E1 -9401.797,E2 -9401.797} C_VEL
LIN {X 0,Y 432.335,Z 296.629,A -85,B 0,C 180,E1 -9404.347,E2 -9404.347} C_VEL
LIN {X 0,Y 432.322,Z 296.633,A -85,B 0,C 180,E1 -9407.016,E2 -9407.016} C_VEL
LIN {X 0,Y 432.335,Z 296.632,A -85,B 0,C 180,E1 -9409.821,E2 -9409.821} C_VEL
LIN {X 0,Y 432.308,Z 296.636,A -85,B 0,C 180,E1 -9413.022,E2 -9413.022} C_VEL
LIN {X 0,Y 432.362,Z 296.634,A -85,B 0,C 180,E1 -9415.996,E2 -9415.996} C_VEL
LIN {X 0,Y 432.35,Z 296.633,A -85,B 0,C 180,E1 -9419.489,E2 -9419.489} C_VEL
LIN {X 0,Y 432.41,Z 296.626,A -85,B 0,C 180,E1 -9423.027,E2 -9423.027} C_VEL
LIN {X 0,Y 434.755,Z 308.374,A -85,B 0,C 180,E1 -9425.401,E2 -9425.401} C_VEL
LIN {X 0,Y 434.977,Z 312.477,A -85,B 0,C 180,E1 -9426.176,E2 -9426.176} C_VEL
LIN {X 0,Y 434.026,Z 331.385,A -85,B 0,C 180,E1 -9429.616,E2 -9429.616} C_VEL
LIN {X 0,Y 433.546,Z 341.438,A -85,B 0,C 180,E1 -9431.425,E2 -9431.425} C_VEL
LIN {X 0,Y 437.389,Z 366.181,A -85,B 0,C 180,E1 -9432.063,E2 -9432.063} C_VEL
LIN {X 0,Y 436.341,Z 450.706,A -85,B 0,C 180,E1 -9433.568,E2 -9433.568} C_VEL
LIN {X 0,Y 435.874,Z 463.67,A -85,B 0,C 180,E1 -9433.971,E2 -9433.971} C_VEL
LIN {X 0,Y 435.246,Z 476.298,A -85,B 0,C 180,E1 -9434.548,E2 -9434.548} C_VEL
LIN {X 0,Y 434.66,Z 487.61,A -85,B 0,C 180,E1 -9435.246,E2 -9435.246} C_VEL
LIN {X 0,Y 434.037,Z 498.664,A -85,B 0,C 180,E1 -9436.12,E2 -9436.12} C_VEL
LIN {X 0,Y 433.347,Z 509.9,A -85,B 0,C 180,E1 -9437.234,E2 -9437.234} C_VEL
LIN {X 0,Y 432.779,Z 518.549,A -85,B 0,C 180,E1 -9438.288,E2 -9438.288} C_VEL
LIN {X 0,Y 432.224,Z 526.533,A -85,B 0,C 180,E1 -9439.459,E2 -9439.459} C_VEL
LIN {X 0,Y 431.789,Z 534.336,A -85,B 0,C 180,E1 -9440.868,E2 -9440.868} C_VEL
LIN {X 0,Y 431.491,Z 541.535,A -85,B 0,C 180,E1 -9442.512,E2 -9442.512} C_VEL
LIN {X 0,Y 431.28,Z 546.651,A -85,B 0,C 180,E1 -9444.024,E2 -9444.024} C_VEL
LIN {X 0,Y 431.27,Z 549.991,A -85,B 0,C 180,E1 -9445.326,E2 -9445.326} C_VEL
LIN {X 0,Y 431.189,Z 551.875,A -85,B 0,C 180,E1 -9446.261,E2 -9446.261} C_VEL
LIN {X 0,Y 431.237,Z 553.292,A -85,B 0,C 180,E1 -9447.197,E2 -9447.197} C_VEL
LIN {X 0,Y 431.218,Z 554.304,A -85,B 0,C 180,E1 -9448.132,E2 -9448.132} C_VEL
LIN {X 0,Y 431.192,Z 554.921,A -85,B 0,C 180,E1 -9449.066,E2 -9449.066} C_VEL
LIN {X 0,Y 431.194,Z 555.124,A -85,B 0,C 180,E1 -9449.999,E2 -9449.999} C_VEL
LIN {X 0,Y 431.192,Z 554.892,A -85,B 0,C 180,E1 -9450.933,E2 -9450.933} C_VEL
LIN {X 0,Y 431.218,Z 554.267,A -85,B 0,C 180,E1 -9451.867,E2 -9451.867} C_VEL
LIN {X 0,Y 431.237,Z 553.246,A -85,B 0,C 180,E1 -9452.802,E2 -9452.802} C_VEL
LIN {X 0,Y 431.19,Z 551.786,A -85,B 0,C 180,E1 -9453.738,E2 -9453.738} C_VEL
LIN {X 0,Y 431.293,Z 548.773,A -85,B 0,C 180,E1 -9455.141,E2 -9455.141} C_VEL
LIN {X 0,Y 431.375,Z 544.682,A -85,B 0,C 180,E1 -9456.548,E2 -9456.548} C_VEL
LIN {X 0,Y 431.601,Z 538.383,A -85,B 0,C 180,E1 -9458.191,E2 -9458.191} C_VEL
LIN {X 0,Y 431.911,Z 531.516,A -85,B 0,C 180,E1 -9459.6,E2 -9459.6} C_VEL
LIN {X 0,Y 432.407,Z 522.954,A -85,B 0,C 180,E1 -9461.009,E2 -9461.009} C_VEL
LIN {X 0,Y 432.987,Z 514.14,A -85,B 0,C 180,E1 -9462.181,E2 -9462.181} C_VEL
LIN {X 0,Y 433.613,Z 503.716,A -85,B 0,C 180,E1 -9463.31,E2 -9463.31} C_VEL
LIN {X 0,Y 434.169,Z 492.428,A -85,B 0,C 180,E1 -9464.291,E2 -9464.291} C_VEL
LIN {X 0,Y 434.85,Z 480.262,A -85,B 0,C 180,E1 -9465.106,E2 -9465.106} C_VEL
LIN {X 0,Y 435.479,Z 467.59,A -85,B 0,C 180,E1 -9465.743,E2 -9465.743} C_VEL
LIN {X 0,Y 435.927,Z 455.169,A -85,B 0,C 180,E1 -9466.176,E2 -9466.176} C_VEL
LIN {X 0,Y 436.234,Z 437.983,A -85,B 0,C 180,E1 -9466.525,E2 -9466.525} C_VEL
LIN {X 0,Y 437.035,Z 366.439,A -85,B 0,C 180,E1 -9467.763,E2 -9467.763} C_VEL
LIN {X 0,Y 433.474,Z 342.602,A -85,B 0,C 180,E1 -9468.356,E2 -9468.356} C_VEL
LIN {X 0,Y 434.375,Z 326.648,A -85,B 0,C 180,E1 -9471.348,E2 -9471.348} C_VEL
LIN {X 0,Y 435.254,Z 312.369,A -85,B 0,C 180,E1 -9474.06,E2 -9474.06} C_VEL
LIN {X 0,Y 434.256,Z 305.595,A -85,B 0,C 180,E1 -9475.436,E2 -9475.436} C_VEL
LIN {X 0,Y 432.443,Z 296.62,A -85,B 0,C 180,E1 -9477.329,E2 -9477.329} C_VEL
LIN {X 0,Y 432.346,Z 296.628,A -85,B 0,C 180,E1 -9480.51,E2 -9480.51} C_VEL
LIN {X 0,Y 432.357,Z 296.629,A -85,B 0,C 180,E1 -9484.003,E2 -9484.003} C_VEL
LIN {X 0,Y 432.319,Z 296.628,A -85,B 0,C 180,E1 -9487.196,E2 -9487.196} C_VEL
LIN {X 0,Y 432.321,Z 296.634,A -85,B 0,C 180,E1 -9490.56,E2 -9490.56} C_VEL
LIN {X 0,Y 432.314,Z 296.63,A -85,B 0,C 180,E1 -9493.06,E2 -9493.06} C_VEL
LIN {X 0,Y 432.337,Z 296.626,A -85,B 0,C 180,E1 -9495.663,E2 -9495.663} C_VEL
LIN {X 0,Y 432.33,Z 296.633,A -85,B 0,C 180,E1 -9498.397,E2 -9498.397} C_VEL
LIN {X 0,Y 432.343,Z 296.626,A -85,B 0,C 180,E1 -9501.851,E2 -9501.851} C_VEL
LIN {X 0,Y 432.336,Z 296.628,A -85,B 0,C 180,E1 -9505.323,E2 -9505.323} C_VEL
LIN {X 0,Y 432.317,Z 296.634,A -85,B 0,C 180,E1 -9508.654,E2 -9508.654} C_VEL
LIN {X 0,Y 432.376,Z 296.621,A -85,B 0,C 180,E1 -9511.876,E2 -9511.876} C_VEL
LIN {X 0,Y 432.346,Z 296.633,A -85,B 0,C 180,E1 -9514.999,E2 -9514.999} C_VEL
LIN {X 0,Y 432.352,Z 296.624,A -85,B 0,C 180,E1 -9518.046,E2 -9518.046} C_VEL
LIN {X 0,Y 432.38,Z 296.627,A -85,B 0,C 180,E1 -9521.029,E2 -9521.029} C_VEL
LIN {X 0,Y 432.425,Z 296.616,A -85,B 0,C 180,E1 -9523.961,E2 -9523.961} C_VEL
LIN {X 0,Y 432.453,Z 296.615,A -85,B 0,C 180,E1 -9527.803,E2 -9527.803} C_VEL
LIN {X 0,Y 432.486,Z 296.615,A -85,B 0,C 180,E1 -9531.59,E2 -9531.59} C_VEL
LIN {X 0,Y 432.591,Z 296.595,A -85,B 0,C 180,E1 -9534.406,E2 -9534.406} C_VEL
LIN {X 0,Y 432.597,Z 296.596,A -85,B 0,C 180,E1 -9538.138,E2 -9538.138} C_VEL
LIN {X 0,Y 432.725,Z 296.582,A -85,B 0,C 180,E1 -9540,E2 -9540} C_VEL
LIN {X 0,Y 432.587,Z 296.595,A -85,B 0,C 180,E1 -9542.794,E2 -9542.794} C_VEL
LIN {X 0,Y 432.58,Z 296.6,A -85,B 0,C 180,E1 -9545.594,E2 -9545.594} C_VEL
LIN {X 0,Y 432.477,Z 296.611,A -85,B 0,C 180,E1 -9548.41,E2 -9548.41} C_VEL
LIN {X 0,Y 432.454,Z 296.618,A -85,B 0,C 180,E1 -9552.197,E2 -9552.197} C_VEL
LIN {X 0,Y 432.424,Z 296.622,A -85,B 0,C 180,E1 -9556.039,E2 -9556.039} C_VEL
LIN {X 0,Y 432.381,Z 296.621,A -85,B 0,C 180,E1 -9559.486,E2 -9559.486} C_VEL
LIN {X 0,Y 432.312,Z 296.63,A -85,B 0,C 180,E1 -9562.965,E2 -9562.965} C_VEL
LIN {X 0,Y 432.334,Z 296.628,A -85,B 0,C 180,E1 -9565.003,E2 -9565.003} C_VEL
LIN {X 0,Y 432.343,Z 296.629,A -85,B 0,C 180,E1 -9568.127,E2 -9568.127} C_VEL
LIN {X 0,Y 432.317,Z 296.629,A -85,B 0,C 180,E1 -9571.347,E2 -9571.347} C_VEL
LIN {X 0,Y 432.336,Z 296.635,A -85,B 0,C 180,E1 -9574.678,E2 -9574.678} C_VEL
LIN {X 0,Y 432.329,Z 296.628,A -85,B 0,C 180,E1 -9578.151,E2 -9578.151} C_VEL
LIN {X 0,Y 432.322,Z 296.629,A -85,B 0,C 180,E1 -9581.602,E2 -9581.602} C_VEL
LIN {X 0,Y 432.331,Z 296.628,A -85,B 0,C 180,E1 -9584.348,E2 -9584.348} C_VEL
LIN {X 0,Y 432.305,Z 296.639,A -85,B 0,C 180,E1 -9587.019,E2 -9587.019} C_VEL
LIN {X 0,Y 432.307,Z 296.63,A -85,B 0,C 180,E1 -9589.826,E2 -9589.826} C_VEL
LIN {X 0,Y 432.305,Z 296.637,A -85,B 0,C 180,E1 -9593.023,E2 -9593.023} C_VEL
LIN {X 0,Y 432.358,Z 296.624,A -85,B 0,C 180,E1 -9595.998,E2 -9595.998} C_VEL
LIN {X 0,Y 432.344,Z 296.632,A -85,B 0,C 180,E1 -9599.492,E2 -9599.492} C_VEL
LIN {X 0,Y 432.328,Z 296.63,A -85,B 0,C 180,E1 -9601.874,E2 -9601.874} C_VEL
LIN {X 0,Y 432.351,Z 296.632,A -85,B 0,C 180,E1 -9605.548,E2 -9605.548} C_VEL
LIN {X 0,Y 432.352,Z 296.626,A -85,B 0,C 180,E1 -9609.047,E2 -9609.047} C_VEL
LIN {X 0,Y 432.359,Z 296.627,A -85,B 0,C 180,E1 -9612.011,E2 -9612.011} C_VEL
LIN {X 0,Y 432.392,Z 296.62,A -85,B 0,C 180,E1 -9614.927,E2 -9614.927} C_VEL
LIN {X 0,Y 432.457,Z 296.619,A -85,B 0,C 180,E1 -9617.804,E2 -9617.804} C_VEL
LIN {X 0,Y 432.449,Z 296.616,A -85,B 0,C 180,E1 -9621.59,E2 -9621.59} C_VEL
LIN {X 0,Y 432.554,Z 296.602,A -85,B 0,C 180,E1 -9624.406,E2 -9624.406} C_VEL
LIN {X 0,Y 432.595,Z 296.602,A -85,B 0,C 180,E1 -9628.139,E2 -9628.139} C_VEL
LIN {X 0,Y 432.624,Z 296.596,A -85,B 0,C 180,E1 -9630.001,E2 -9630.001} C_VEL
LIN {X 0,Y 432.542,Z 296.602,A -85,B 0,C 180,E1 -9632.794,E2 -9632.794} C_VEL
LIN {X 0,Y 432.426,Z 296.616,A -85,B 0,C 180,E1 -9635.013,E2 -9635.013} C_VEL
LIN {X 0,Y 431.856,Z 296.689,A -85,B 0,C 180,E1 -9635.791,E2 -9635.791} C_VEL
LIN {X 0,Y 429.004,Z 297.043,A -85,B 0,C 180,E1 -9637.056,E2 -9637.056} C_VEL
LIN {X 0,Y 426.526,Z 297.354,A -85,B 0,C 180,E1 -9638.076,E2 -9638.076} C_VEL
LIN {X 0,Y 425.457,Z 297.487,A -85,B 0,C 180,E1 -9638.866,E2 -9638.866} C_VEL
LIN {X 0,Y 425.371,Z 297.495,A -85,B 0,C 180,E1 -9639.134,E2 -9639.134} C_VEL
LIN {X 0,Y 425.389,Z 297.495,A -85,B 0,C 180,E1 -9642.898,E2 -9642.898} C_VEL
LIN {X 0,Y 425.322,Z 297.508,A -85,B 0,C 180,E1 -9646.585,E2 -9646.585} C_VEL
LIN {X 0,Y 425.301,Z 297.503,A -85,B 0,C 180,E1 -9649.623,E2 -9649.623} C_VEL
LIN {X 0,Y 425.289,Z 297.51,A -85,B 0,C 180,E1 -9652.339,E2 -9652.339} C_VEL
LIN {X 0,Y 425.34,Z 297.7,A -85,B 0,C 180,E1 -9654.996,E2 -9654.996} C_VEL
LIN {X 0,Y 426.977,Z 307.183,A -85,B 0,C 180,E1 -9657.272,E2 -9657.272} C_VEL
LIN {X 0,Y 426.786,Z 312.459,A -85,B 0,C 180,E1 -9658.459,E2 -9658.459} C_VEL
LIN {X 0,Y 430.456,Z 331.611,A -85,B 0,C 180,E1 -9658.97,E2 -9658.97} C_VEL
LIN {X 0,Y 429.321,Z 420.002,A -85,B 0,C 180,E1 -9660.547,E2 -9660.547} C_VEL
LIN {X 0,Y 428.865,Z 433.819,A -85,B 0,C 180,E1 -9660.993,E2 -9660.993} C_VEL
LIN {X 0,Y 428.468,Z 446.337,A -85,B 0,C 180,E1 -9661.597,E2 -9661.597} C_VEL
LIN {X 0,Y 427.826,Z 458.716,A -85,B 0,C 180,E1 -9662.408,E2 -9662.408} C_VEL
LIN {X 0,Y 427.196,Z 469.728,A -85,B 0,C 180,E1 -9663.332,E2 -9663.332} C_VEL
LIN {X 0,Y 426.617,Z 480.388,A -85,B 0,C 180,E1 -9664.458,E2 -9664.458} C_VEL
LIN {X 0,Y 426.048,Z 488.747,A -85,B 0,C 180,E1 -9665.537,E2 -9665.537} C_VEL
LIN {X 0,Y 425.404,Z 497.908,A -85,B 0,C 180,E1 -9666.992,E2 -9666.992} C_VEL
LIN {X 0,Y 424.978,Z 504.687,A -85,B 0,C 180,E1 -9668.327,E2 -9668.327} C_VEL
LIN {X 0,Y 424.653,Z 510.992,A -85,B 0,C 180,E1 -9669.89,E2 -9669.89} C_VEL
LIN {X 0,Y 424.383,Z 515.917,A -85,B 0,C 180,E1 -9671.485,E2 -9671.485} C_VEL
LIN {X 0,Y 424.198,Z 519.741,A -85,B 0,C 180,E1 -9673.198,E2 -9673.198} C_VEL
LIN {X 0,Y 424.053,Z 521.735,A -85,B 0,C 180,E1 -9674.548,E2 -9674.548} C_VEL
LIN {X 0,Y 424.002,Z 522.896,A -85,B 0,C 180,E1 -9675.879,E2 -9675.879} C_VEL
LIN {X 0,Y 423.991,Z 523.285,A -85,B 0,C 180,E1 -9677.186,E2 -9677.186} C_VEL
LIN {X 0,Y 424.035,Z 522.893,A -85,B 0,C 180,E1 -9678.473,E2 -9678.473} C_VEL
LIN {X 0,Y 424.041,Z 521.799,A -85,B 0,C 180,E1 -9679.73,E2 -9679.73} C_VEL
LIN {X 0,Y 424.204,Z 519.725,A -85,B 0,C 180,E1 -9681.14,E2 -9681.14} C_VEL
LIN {X 0,Y 424.422,Z 516.464,A -85,B 0,C 180,E1 -9682.64,E2 -9682.64} C_VEL
LIN {X 0,Y 424.712,Z 511.901,A -85,B 0,C 180,E1 -9684.178,E2 -9684.178} C_VEL
LIN {X 0,Y 425.109,Z 505.623,A -85,B 0,C 180,E1 -9685.799,E2 -9685.799} C_VEL
LIN {X 0,Y 425.657,Z 497.806,A -85,B 0,C 180,E1 -9687.358,E2 -9687.358} C_VEL
LIN {X 0,Y 426.216,Z 490.086,A -85,B 0,C 180,E1 -9688.602,E2 -9688.602} C_VEL
LIN {X 0,Y 426.903,Z 480.54,A -85,B 0,C 180,E1 -9689.86,E2 -9689.86} C_VEL
LIN {X 0,Y 427.589,Z 469.742,A -85,B 0,C 180,E1 -9690.995,E2 -9690.995} C_VEL
LIN {X 0,Y 428.33,Z 457.719,A -85,B 0,C 180,E1 -9691.994,E2 -9691.994} C_VEL
LIN {X 0,Y 428.908,Z 446.966,A -85,B 0,C 180,E1 -9692.69,E2 -9692.69} C_VEL
LIN {X 0,Y 429.353,Z 433.72,A -85,B 0,C 180,E1 -9693.329,E2 -9693.329} C_VEL
LIN {X 0,Y 429.718,Z 421.466,A -85,B 0,C 180,E1 -9693.729,E2 -9693.729} C_VEL
LIN {X 0,Y 430.542,Z 363.822,A -85,B 0,C 180,E1 -9694.788,E2 -9694.788} C_VEL
LIN {X 0,Y 431.033,Z 330.914,A -85,B 0,C 180,E1 -9695.381,E2 -9695.381} C_VEL
LIN {X 0,Y 427.156,Z 311.883,A -85,B 0,C 180,E1 -9695.97,E2 -9695.97} C_VEL
LIN {X 0,Y 427.087,Z 305.658,A -85,B 0,C 180,E1 -9697.149,E2 -9697.149} C_VEL
LIN {X 0,Y 425.315,Z 297.509,A -85,B 0,C 180,E1 -9698.809,E2 -9698.809} C_VEL
LIN {X 0,Y 425.332,Z 297.508,A -85,B 0,C 180,E1 -9701.702,E2 -9701.702} C_VEL
LIN {X 0,Y 425.351,Z 297.504,A -85,B 0,C 180,E1 -9704.67,E2 -9704.67} C_VEL
LIN {X 0,Y 425.414,Z 297.497,A -85,B 0,C 180,E1 -9707.598,E2 -9707.598} C_VEL
LIN {X 0,Y 425.444,Z 297.491,A -85,B 0,C 180,E1 -9711.45,E2 -9711.45} C_VEL
LIN {X 0,Y 425.552,Z 297.476,A -85,B 0,C 180,E1 -9714.313,E2 -9714.313} C_VEL
LIN {X 0,Y 425.574,Z 297.473,A -85,B 0,C 180,E1 -9718.107,E2 -9718.107} C_VEL
LIN {X 0,Y 425.703,Z 297.459,A -85,B 0,C 180,E1 -9720,E2 -9720} C_VEL
LIN {X 0,Y 425.547,Z 297.474,A -85,B 0,C 180,E1 -9722.84,E2 -9722.84} C_VEL
LIN {X 0,Y 425.542,Z 297.477,A -85,B 0,C 180,E1 -9725.687,E2 -9725.687} C_VEL
LIN {X 0,Y 425.438,Z 297.49,A -85,B 0,C 180,E1 -9728.55,E2 -9728.55} C_VEL
LIN {X 0,Y 425.414,Z 297.494,A -85,B 0,C 180,E1 -9732.402,E2 -9732.402} C_VEL
LIN {X 0,Y 425.389,Z 297.497,A -85,B 0,C 180,E1 -9736.312,E2 -9736.312} C_VEL
LIN {X 0,Y 425.33,Z 297.5,A -85,B 0,C 180,E1 -9739.635,E2 -9739.635} C_VEL
LIN {X 0,Y 425.289,Z 297.507,A -85,B 0,C 180,E1 -9742.339,E2 -9742.339} C_VEL
LIN {X 0,Y 425.297,Z 297.504,A -85,B 0,C 180,E1 -9745.445,E2 -9745.445} C_VEL
LIN {X 0,Y 425.333,Z 297.499,A -85,B 0,C 180,E1 -9748.632,E2 -9748.632} C_VEL
LIN {X 0,Y 425.266,Z 297.506,A -85,B 0,C 180,E1 -9751.927,E2 -9751.927} C_VEL
LIN {X 0,Y 425.299,Z 297.508,A -85,B 0,C 180,E1 -9755.336,E2 -9755.336} C_VEL
LIN {X 0,Y 425.303,Z 297.506,A -85,B 0,C 180,E1 -9758.898,E2 -9758.898} C_VEL
LIN {X 0,Y 425.292,Z 297.508,A -85,B 0,C 180,E1 -9761.958,E2 -9761.958} C_VEL
LIN {X 0,Y 425.286,Z 297.512,A -85,B 0,C 180,E1 -9765.283,E2 -9765.283} C_VEL
LIN {X 0,Y 425.276,Z 297.508,A -85,B 0,C 180,E1 -9768.621,E2 -9768.621} C_VEL
LIN {X 0,Y 425.299,Z 297.508,A -85,B 0,C 180,E1 -9771.101,E2 -9771.101} C_VEL
LIN {X 0,Y 425.302,Z 297.509,A -85,B 0,C 180,E1 -9774.664,E2 -9774.664} C_VEL
LIN {X 0,Y 425.268,Z 297.517,A -85,B 0,C 180,E1 -9778.073,E2 -9778.073} C_VEL
LIN {X 0,Y 425.334,Z 297.505,A -85,B 0,C 180,E1 -9781.368,E2 -9781.368} C_VEL
LIN {X 0,Y 425.383,Z 297.592,A -85,B 0,C 180,E1 -9782.783,E2 -9782.783} C_VEL
LIN {X 0,Y 427.821,Z 309.574,A -85,B 0,C 180,E1 -9785.236,E2 -9785.236} C_VEL
LIN {X 0,Y 428.081,Z 313.669,A -85,B 0,C 180,E1 -9786.025,E2 -9786.025} C_VEL
LIN {X 0,Y 427.066,Z 332.805,A -85,B 0,C 180,E1 -9789.556,E2 -9789.556} C_VEL
LIN {X 0,Y 426.638,Z 341.141,A -85,B 0,C 180,E1 -9791.084,E2 -9791.084} C_VEL
LIN {X 0,Y 430.627,Z 366.56,A -85,B 0,C 180,E1 -9791.761,E2 -9791.761} C_VEL
LIN {X 0,Y 429.57,Z 451.082,A -85,B 0,C 180,E1 -9793.301,E2 -9793.301} C_VEL
LIN {X 0,Y 429.071,Z 463.822,A -85,B 0,C 180,E1 -9793.709,E2 -9793.709} C_VEL
LIN {X 0,Y 428.417,Z 476.334,A -85,B 0,C 180,E1 -9794.295,E2 -9794.295} C_VEL
LIN {X 0,Y 427.784,Z 487.546,A -85,B 0,C 180,E1 -9795.003,E2 -9795.003} C_VEL
LIN {X 0,Y 427.123,Z 498.758,A -85,B 0,C 180,E1 -9795.911,E2 -9795.911} C_VEL
LIN {X 0,Y 426.363,Z 509.733,A -85,B 0,C 180,E1 -9797.021,E2 -9797.021} C_VEL
LIN {X 0,Y 425.794,Z 518.354,A -85,B 0,C 180,E1 -9798.093,E2 -9798.093} C_VEL
LIN {X 0,Y 425.221,Z 526.319,A -85,B 0,C 180,E1 -9799.284,E2 -9799.284} C_VEL
LIN {X 0,Y 424.744,Z 534.111,A -85,B 0,C 180,E1 -9800.716,E2 -9800.716} C_VEL
LIN {X 0,Y 424.518,Z 539.457,A -85,B 0,C 180,E1 -9801.91,E2 -9801.91} C_VEL
LIN {X 0,Y 424.299,Z 544.634,A -85,B 0,C 180,E1 -9803.341,E2 -9803.341} C_VEL
LIN {X 0,Y 424.206,Z 548.657,A -85,B 0,C 180,E1 -9804.771,E2 -9804.771} C_VEL
LIN {X 0,Y 424.1,Z 551.628,A -85,B 0,C 180,E1 -9806.199,E2 -9806.199} C_VEL
LIN {X 0,Y 424.133,Z 553.04,A -85,B 0,C 180,E1 -9807.15,E2 -9807.15} C_VEL
LIN {X 0,Y 424.143,Z 554.05,A -85,B 0,C 180,E1 -9808.1,E2 -9808.1} C_VEL
LIN {X 0,Y 424.111,Z 554.664,A -85,B 0,C 180,E1 -9809.05,E2 -9809.05} C_VEL
LIN {X 0,Y 424.109,Z 554.856,A -85,B 0,C 180,E1 -9809.999,E2 -9809.999} C_VEL
LIN {X 0,Y 424.111,Z 554.618,A -85,B 0,C 180,E1 -9810.949,E2 -9810.949} C_VEL
LIN {X 0,Y 424.143,Z 553.988,A -85,B 0,C 180,E1 -9811.899,E2 -9811.899} C_VEL
LIN {X 0,Y 424.134,Z 552.959,A -85,B 0,C 180,E1 -9812.849,E2 -9812.849} C_VEL
LIN {X 0,Y 424.101,Z 551.485,A -85,B 0,C 180,E1 -9813.8,E2 -9813.8} C_VEL
LIN {X 0,Y 424.205,Z 548.455,A -85,B 0,C 180,E1 -9815.228,E2 -9815.228} C_VEL
LIN {X 0,Y 424.298,Z 544.345,A -85,B 0,C 180,E1 -9816.658,E2 -9816.658} C_VEL
LIN {X 0,Y 424.533,Z 538.023,A -85,B 0,C 180,E1 -9818.328,E2 -9818.328} C_VEL
LIN {X 0,Y 424.881,Z 531.131,A -85,B 0,C 180,E1 -9819.761,E2 -9819.761} C_VEL
LIN {X 0,Y 425.291,Z 524.094,A -85,B 0,C 180,E1 -9820.954,E2 -9820.954} C_VEL
LIN {X 0,Y 425.897,Z 515.62,A -85,B 0,C 180,E1 -9822.145,E2 -9822.145} C_VEL
LIN {X 0,Y 426.468,Z 506.329,A -85,B 0,C 180,E1 -9823.217,E2 -9823.217} C_VEL
LIN {X 0,Y 427.106,Z 494.781,A -85,B 0,C 180,E1 -9824.289,E2 -9824.289} C_VEL
LIN {X 0,Y 427.756,Z 483.455,A -85,B 0,C 180,E1 -9825.118,E2 -9825.118} C_VEL
LIN {X 0,Y 428.373,Z 471.953,A -85,B 0,C 180,E1 -9825.766,E2 -9825.766} C_VEL
LIN {X 0,Y 428.888,Z 458.829,A -85,B 0,C 180,E1 -9826.297,E2 -9826.297} C_VEL
LIN {X 0,Y 429.256,Z 446.375,A -85,B 0,C 180,E1 -9826.618,E2 -9826.618} C_VEL
LIN {X 0,Y 430.19,Z 366.842,A -85,B 0,C 180,E1 -9828.022,E2 -9828.022} C_VEL
LIN {X 0,Y 426.503,Z 342.368,A -85,B 0,C 180,E1 -9828.642,E2 -9828.642} C_VEL
LIN {X 0,Y 427.474,Z 326.305,A -85,B 0,C 180,E1 -9831.71,E2 -9831.71} C_VEL
LIN {X 0,Y 428.32,Z 313.324,A -85,B 0,C 180,E1 -9834.217,E2 -9834.217} C_VEL
LIN {X 0,Y 426.743,Z 304.105,A -85,B 0,C 180,E1 -9836.138,E2 -9836.138} C_VEL
LIN {X 0,Y 425.388,Z 297.498,A -85,B 0,C 180,E1 -9837.587,E2 -9837.587} C_VEL
LIN {X 0,Y 425.286,Z 297.505,A -85,B 0,C 180,E1 -9840.815,E2 -9840.815} C_VEL
LIN {X 0,Y 425.309,Z 297.509,A -85,B 0,C 180,E1 -9844.287,E2 -9844.287} C_VEL
LIN {X 0,Y 425.275,Z 297.507,A -85,B 0,C 180,E1 -9847.694,E2 -9847.694} C_VEL
LIN {X 0,Y 425.276,Z 297.512,A -85,B 0,C 180,E1 -9850.52,E2 -9850.52} C_VEL
LIN {X 0,Y 425.254,Z 297.509,A -85,B 0,C 180,E1 -9853.35,E2 -9853.35} C_VEL
LIN {X 0,Y 425.26,Z 297.515,A -85,B 0,C 180,E1 -9856.647,E2 -9856.647} C_VEL
LIN {X 0,Y 425.291,Z 297.505,A -85,B 0,C 180,E1 -9859.873,E2 -9859.873} C_VEL
LIN {X 0,Y 425.28,Z 297.511,A -85,B 0,C 180,E1 -9862.487,E2 -9862.487} C_VEL
LIN {X 0,Y 425.303,Z 297.502,A -85,B 0,C 180,E1 -9865.817,E2 -9865.817} C_VEL
LIN {X 0,Y 425.285,Z 297.508,A -85,B 0,C 180,E1 -9869.238,E2 -9869.238} C_VEL
LIN {X 0,Y 425.343,Z 297.499,A -85,B 0,C 180,E1 -9872.442,E2 -9872.442} C_VEL
LIN {X 0,Y 425.346,Z 297.499,A -85,B 0,C 180,E1 -9875.602,E2 -9875.602} C_VEL
LIN {X 0,Y 425.287,Z 297.507,A -85,B 0,C 180,E1 -9878.681,E2 -9878.681} C_VEL
LIN {X 0,Y 425.327,Z 297.502,A -85,B 0,C 180,E1 -9881.703,E2 -9881.703} C_VEL
LIN {X 0,Y 425.343,Z 297.499,A -85,B 0,C 180,E1 -9884.671,E2 -9884.671} C_VEL
LIN {X 0,Y 425.406,Z 297.495,A -85,B 0,C 180,E1 -9887.598,E2 -9887.598} C_VEL
LIN {X 0,Y 425.436,Z 297.494,A -85,B 0,C 180,E1 -9891.45,E2 -9891.45} C_VEL
LIN {X 0,Y 425.548,Z 297.473,A -85,B 0,C 180,E1 -9894.313,E2 -9894.313} C_VEL
LIN {X 0,Y 425.566,Z 297.472,A -85,B 0,C 180,E1 -9898.107,E2 -9898.107} C_VEL
LIN {X 0,Y 425.695,Z 297.458,A -85,B 0,C 180,E1 -9900,E2 -9900} C_VEL
LIN {X 0,Y 425.541,Z 297.473,A -85,B 0,C 180,E1 -9902.84,E2 -9902.84} C_VEL
LIN {X 0,Y 425.491,Z 297.479,A -85,B 0,C 180,E1 -9906.521,E2 -9906.521} C_VEL
LIN {X 0,Y 425.395,Z 297.493,A -85,B 0,C 180,E1 -9909.51,E2 -9909.51} C_VEL
LIN {X 0,Y 425.388,Z 297.492,A -85,B 0,C 180,E1 -9912.904,E2 -9912.904} C_VEL
LIN {X 0,Y 425.355,Z 297.499,A -85,B 0,C 180,E1 -9916.605,E2 -9916.605} C_VEL
LIN {X 0,Y 425.323,Z 297.501,A -85,B 0,C 180,E1 -9919.636,E2 -9919.636} C_VEL
LIN {X 0,Y 425.283,Z 297.513,A -85,B 0,C 180,E1 -9922.339,E2 -9922.339} C_VEL
LIN {X 0,Y 425.316,Z 297.505,A -85,B 0,C 180,E1 -9924.658,E2 -9924.658} C_VEL
LIN {X 0,Y 425.267,Z 297.507,A -85,B 0,C 180,E1 -9927.564,E2 -9927.564} C_VEL
LIN {X 0,Y 425.286,Z 297.51,A -85,B 0,C 180,E1 -9930.762,E2 -9930.762} C_VEL
LIN {X 0,Y 425.308,Z 297.505,A -85,B 0,C 180,E1 -9934.289,E2 -9934.289} C_VEL
LIN {X 0,Y 425.274,Z 297.506,A -85,B 0,C 180,E1 -9937.695,E2 -9937.695} C_VEL
LIN {X 0,Y 425.263,Z 297.512,A -85,B 0,C 180,E1 -9940.519,E2 -9940.519} C_VEL
LIN {X 0,Y 425.253,Z 297.511,A -85,B 0,C 180,E1 -9943.351,E2 -9943.351} C_VEL
LIN {X 0,Y 425.256,Z 297.508,A -85,B 0,C 180,E1 -9946.045,E2 -9946.045} C_VEL
LIN {X 0,Y 425.254,Z 297.512,A -85,B 0,C 180,E1 -9949.485,E2 -9949.485} C_VEL
LIN {X 0,Y 425.276,Z 297.507,A -85,B 0,C 180,E1 -9952.49,E2 -9952.49} C_VEL
LIN {X 0,Y 425.305,Z 297.504,A -85,B 0,C 180,E1 -9955.818,E2 -9955.818} C_VEL
LIN {X 0,Y 425.29,Z 297.511,A -85,B 0,C 180,E1 -9959.24,E2 -9959.24} C_VEL
LIN {X 0,Y 425.305,Z 297.51,A -85,B 0,C 180,E1 -9961.367,E2 -9961.367} C_VEL
LIN {X 0,Y 425.259,Z 297.508,A -85,B 0,C 180,E1 -9964.553,E2 -9964.553} C_VEL
LIN {X 0,Y 425.294,Z 297.51,A -85,B 0,C 180,E1 -9967.731,E2 -9967.731} C_VEL
LIN {X 0,Y 425.363,Z 297.495,A -85,B 0,C 180,E1 -9970.705,E2 -9970.705} C_VEL
LIN {X 0,Y 425.389,Z 297.5,A -85,B 0,C 180,E1 -9973.689,E2 -9973.689} C_VEL
LIN {X 0,Y 425.412,Z 297.494,A -85,B 0,C 180,E1 -9977.599,E2 -9977.599} C_VEL
LIN {X 0,Y 425.397,Z 297.493,A -85,B 0,C 180,E1 -9981.45,E2 -9981.45} C_VEL
LIN {X 0,Y 425.512,Z 297.481,A -85,B 0,C 180,E1 -9984.313,E2 -9984.313} C_VEL
LIN {X 0,Y 425.564,Z 297.478,A -85,B 0,C 180,E1 -9988.108,E2 -9988.108} C_VEL
LIN {X 0,Y 425.576,Z 297.474,A -85,B 0,C 180,E1 -9990.001,E2 -9990.001} C_VEL
LIN {X 0,Y 425.499,Z 297.479,A -85,B 0,C 180,E1 -9992.841,E2 -9992.841} C_VEL
LIN {X 0,Y 425.512,Z 297.478,A -85,B 0,C 180,E1 -9995.688,E2 -9995.688} C_VEL
LIN {X 0,Y 425.397,Z 297.497,A -85,B 0,C 180,E1 -9998.551,E2 -9998.551} C_VEL
LIN {X 0,Y 425.371,Z 297.495,A -85,B 0,C 180,E1 -9999.134,E2 -9999.134} C_VEL
LIN {X 0,Y 424.718,Z 297.579,A -85,B 0,C 180,E1 -9999.924,E2 -9999.924} C_VEL
LIN {X 0,Y 421.896,Z 297.928,A -85,B 0,C 180,E1 -10001.208,E2 -10001.208} C_VEL
LIN {X 0,Y 419.481,Z 298.232,A -85,B 0,C 180,E1 -10002.244,E2 -10002.244} C_VEL
LIN {X 0,Y 418.41,Z 298.364,A -85,B 0,C 180,E1 -10003.045,E2 -10003.045} C_VEL
LIN {X 0,Y 418.305,Z 298.375,A -85,B 0,C 180,E1 -10003.316,E2 -10003.316} C_VEL
LIN {X 0,Y 418.267,Z 298.386,A -85,B 0,C 180,E1 -10006.712,E2 -10006.712} C_VEL
LIN {X 0,Y 418.247,Z 298.382,A -85,B 0,C 180,E1 -10009.779,E2 -10009.779} C_VEL
LIN {X 0,Y 418.229,Z 298.391,A -85,B 0,C 180,E1 -10012.737,E2 -10012.737} C_VEL
LIN {X 0,Y 418.292,Z 298.419,A -85,B 0,C 180,E1 -10014.755,E2 -10014.755} C_VEL
LIN {X 0,Y 420.005,Z 308.401,A -85,B 0,C 180,E1 -10017.187,E2 -10017.187} C_VEL
LIN {X 0,Y 419.894,Z 312.603,A -85,B 0,C 180,E1 -10018.151,E2 -10018.151} C_VEL
LIN {X 0,Y 423.624,Z 331.891,A -85,B 0,C 180,E1 -10018.691,E2 -10018.691} C_VEL
LIN {X 0,Y 422.448,Z 420.769,A -85,B 0,C 180,E1 -10020.314,E2 -10020.314} C_VEL
LIN {X 0,Y 422,Z 434.535,A -85,B 0,C 180,E1 -10020.773,E2 -10020.773} C_VEL
LIN {X 0,Y 421.577,Z 446.905,A -85,B 0,C 180,E1 -10021.387,E2 -10021.387} C_VEL
LIN {X 0,Y 420.926,Z 459.178,A -85,B 0,C 180,E1 -10022.207,E2 -10022.207} C_VEL
LIN {X 0,Y 420.282,Z 469.464,A -85,B 0,C 180,E1 -10023.081,E2 -10023.081} C_VEL
LIN {X 0,Y 419.77,Z 479.323,A -85,B 0,C 180,E1 -10024.117,E2 -10024.117} C_VEL
LIN {X 0,Y 419.083,Z 488.872,A -85,B 0,C 180,E1 -10025.349,E2 -10025.349} C_VEL
LIN {X 0,Y 418.448,Z 497.49,A -85,B 0,C 180,E1 -10026.726,E2 -10026.726} C_VEL
LIN {X 0,Y 417.969,Z 504.511,A -85,B 0,C 180,E1 -10028.11,E2 -10028.11} C_VEL
LIN {X 0,Y 417.589,Z 511.14,A -85,B 0,C 180,E1 -10029.758,E2 -10029.758} C_VEL
LIN {X 0,Y 417.399,Z 515.21,A -85,B 0,C 180,E1 -10031.047,E2 -10031.047} C_VEL
LIN {X 0,Y 417.193,Z 518.453,A -85,B 0,C 180,E1 -10032.364,E2 -10032.364} C_VEL
LIN {X 0,Y 417.029,Z 520.903,A -85,B 0,C 180,E1 -10033.706,E2 -10033.706} C_VEL
LIN {X 0,Y 416.943,Z 522.565,A -85,B 0,C 180,E1 -10035.069,E2 -10035.069} C_VEL
LIN {X 0,Y 416.903,Z 523.433,A -85,B 0,C 180,E1 -10036.459,E2 -10036.459} C_VEL
LIN {X 0,Y 416.901,Z 523.452,A -85,B 0,C 180,E1 -10037.88,E2 -10037.88} C_VEL
LIN {X 0,Y 416.933,Z 522.553,A -85,B 0,C 180,E1 -10039.336,E2 -10039.336} C_VEL
LIN {X 0,Y 417.08,Z 520.692,A -85,B 0,C 180,E1 -10040.817,E2 -10040.817} C_VEL
LIN {X 0,Y 417.354,Z 516.916,A -85,B 0,C 180,E1 -10042.683,E2 -10042.683} C_VEL
LIN {X 0,Y 417.647,Z 512.523,A -85,B 0,C 180,E1 -10044.213,E2 -10044.213} C_VEL
LIN {X 0,Y 418.088,Z 506.19,A -85,B 0,C 180,E1 -10045.897,E2 -10045.897} C_VEL
LIN {X 0,Y 418.59,Z 499.43,A -85,B 0,C 180,E1 -10047.309,E2 -10047.309} C_VEL
LIN {X 0,Y 419.245,Z 490.778,A -85,B 0,C 180,E1 -10048.753,E2 -10048.753} C_VEL
LIN {X 0,Y 419.954,Z 481.372,A -85,B 0,C 180,E1 -10050.023,E2 -10050.023} C_VEL
LIN {X 0,Y 420.681,Z 470.804,A -85,B 0,C 180,E1 -10051.171,E2 -10051.171} C_VEL
LIN {X 0,Y 421.429,Z 459.246,A -85,B 0,C 180,E1 -10052.163,E2 -10052.163} C_VEL
LIN {X 0,Y 422.104,Z 447.489,A -85,B 0,C 180,E1 -10052.951,E2 -10052.951} C_VEL
LIN {X 0,Y 422.587,Z 434.59,A -85,B 0,C 180,E1 -10053.59,E2 -10053.59} C_VEL
LIN {X 0,Y 422.969,Z 422.35,A -85,B 0,C 180,E1 -10054.004,E2 -10054.004} C_VEL
LIN {X 0,Y 423.49,Z 389.618,A -85,B 0,C 180,E1 -10054.635,E2 -10054.635} C_VEL
LIN {X 0,Y 424.313,Z 331.353,A -85,B 0,C 180,E1 -10055.711,E2 -10055.711} C_VEL
LIN {X 0,Y 420.289,Z 312.322,A -85,B 0,C 180,E1 -10056.293,E2 -10056.293} C_VEL
LIN {X 0,Y 420.368,Z 308.244,A -85,B 0,C 180,E1 -10057.071,E2 -10057.071} C_VEL
LIN {X 0,Y 418.272,Z 298.384,A -85,B 0,C 180,E1 -10059.145,E2 -10059.145} C_VEL
LIN {X 0,Y 418.288,Z 298.385,A -85,B 0,C 180,E1 -10062.396,E2 -10062.396} C_VEL
LIN {X 0,Y 418.306,Z 298.384,A -85,B 0,C 180,E1 -10065.403,E2 -10065.403} C_VEL
LIN {X 0,Y 418.317,Z 298.376,A -85,B 0,C 180,E1 -10068.369,E2 -10068.369} C_VEL
LIN {X 0,Y 418.516,Z 298.353,A -85,B 0,C 180,E1 -10072.279,E2 -10072.279} C_VEL
LIN {X 0,Y 418.511,Z 298.354,A -85,B 0,C 180,E1 -10074.217,E2 -10074.217} C_VEL
LIN {X 0,Y 418.544,Z 298.349,A -85,B 0,C 180,E1 -10078.075,E2 -10078.075} C_VEL
LIN {X 0,Y 418.672,Z 298.334,A -85,B 0,C 180,E1 -10080,E2 -10080} C_VEL
LIN {X 0,Y 418.503,Z 298.351,A -85,B 0,C 180,E1 -10082.888,E2 -10082.888} C_VEL
LIN {X 0,Y 418.499,Z 298.355,A -85,B 0,C 180,E1 -10085.783,E2 -10085.783} C_VEL
LIN {X 0,Y 418.398,Z 298.366,A -85,B 0,C 180,E1 -10088.695,E2 -10088.695} C_VEL
LIN {X 0,Y 418.316,Z 298.375,A -85,B 0,C 180,E1 -10091.631,E2 -10091.631} C_VEL
LIN {X 0,Y 418.306,Z 298.38,A -85,B 0,C 180,E1 -10094.597,E2 -10094.597} C_VEL
LIN {X 0,Y 418.281,Z 298.374,A -85,B 0,C 180,E1 -10097.604,E2 -10097.604} C_VEL
